(* IEC 61131-3 sources: 5GE_TP_M5/, 10 files *)

(* ---- System_Configuration.st ---- *)
(*
===============================================================================
系统配置和初始化模块
===============================================================================
功能描述：
- 系统参数配置
- I/O地址定义和映射
- 全局变量定义
- 系统常量定义
- 启动序列管理
- 系统自检功能

配置内容：
1. 硬件配置参数
2. 安全参数设置
3. 时间参数配置
4. 密码和权限设置
5. 通信参数配置
6. 诊断参数设置

使用说明：
本文件包含了系统的所有配置参数，在实际部署时需要根据
现场情况调整相关参数。所有参数都有详细说明和推荐值。

作者: Claude Code Assistant
日期: 2025-09-23
版本: 1.0
===============================================================================
*)

(*  ============================================================================ *)
(*  全局变量定义（用于Unity Pro全局变量表） *)
(*  ============================================================================ *)

VAR_GLOBAL
    (*  ======================================================================== *)
    (*  系统配置参数 *)
    (*  ======================================================================== *)
    CFG_System_Version      : STRING[10] := '1.0.0';    (*  系统版本号 *)
    CFG_PLC_Model           : STRING[20] := 'BMX P34 20102 V2.10'; (*  PLC型号 *)
    CFG_Project_Name        : STRING[30] := 'Dual_Gate_Control_System'; (*  项目名称 *)
    CFG_Installation_Date   : STRING[10] := '2025-09-23'; (*  安装日期 *)
    CFG_Commissioning_Date  : STRING[10] := '2025-09-23'; (*  调试日期 *)

    (*  ======================================================================== *)
    (*  硬件配置参数 *)
    (*  ======================================================================== *)
    CFG_Gate1_Type          : STRING[15] := 'Swing_Panel';     (*  门板1类型 *)
    CFG_Gate2_Type          : STRING[15] := 'Swing_Panel';     (*  门板2类型 *)
    CFG_Motor_Power         : REAL := 0.5;           (*  电机功率 (kW) *)
    CFG_Gate_Weight         : REAL := 150.0;         (*  门板重量 (kg) *)
    CFG_Gate_Width          : REAL := 1.5;           (*  门板宽度 (m) *)

    (*  ======================================================================== *)
    (*  安全参数配置 *)
    (*  ======================================================================== *)
    CFG_Max_Opening_Time    : TIME := T#30s;         (*  最大开门时间 *)
    CFG_Max_Closing_Time    : TIME := T#30s;         (*  最大关门时间 *)
    CFG_Obstacle_Delay      : TIME := T#1s;          (*  障碍物检测延时 *)
    CFG_Overcurrent_Delay   : TIME := T#500ms;       (*  过流检测延时 *)
    CFG_Reverse_Duration    : TIME := T#3s;          (*  反向动作持续时间 *)
    CFG_Safety_Reset_Time   : TIME := T#2s;          (*  安全复位时间 *)

    (*  ======================================================================== *)
    (*  控制参数配置 *)
    (*  ======================================================================== *)
    CFG_Command_Timeout     : TIME := T#2s;          (*  命令超时时间 *)
    CFG_Double_Click_Time   : TIME := T#1s;          (*  双击检测时间 *)
    CFG_Intercom_Priority   : BOOL := TRUE;          (*  对讲机优先级 *)
    CFG_Auto_Close_Enable   : BOOL := FALSE;         (*  自动关门使能 *)
    CFG_Auto_Close_Delay    : TIME := T#10s;         (*  自动关门延时 *)

    (*  ======================================================================== *)
    (*  密码和权限配置 *)
    (*  ======================================================================== *)
    CFG_Password_Single     : INT := 1504;           (*  单门密码 *)
    CFG_Password_Dual       : INT := 2502;           (*  双门密码 *)
    CFG_Input_Timeout       : TIME := T#10s;         (*  密码输入超时 *)
    CFG_Valid_Duration      : TIME := T#30s;         (*  密码有效持续时间 *)
    CFG_Lock_Duration       : TIME := T#5m;          (*  锁定持续时间 *)
    CFG_Max_Attempts        : INT := 3;              (*  最大尝试次数 *)

    (*  ======================================================================== *)
    (*  照明和信号配置 *)
    (*  ======================================================================== *)
    CFG_Lighting_Delay      : TIME := T#5m;          (*  照明延时关闭时间 *)
    CFG_Warning_Blink_Cycle : TIME := T#500ms;       (*  警告灯闪烁周期 *)
    CFG_Night_Lighting      : BOOL := TRUE;          (*  夜间照明使能 *)
    CFG_Night_Start_Hour    : INT := 18;             (*  夜间开始时间 *)
    CFG_Night_End_Hour      : INT := 6;              (*  夜间结束时间 *)

    (*  ======================================================================== *)
    (*  通信配置参数 *)
    (*  ======================================================================== *)
    CFG_Ethernet_IP         : STRING[15] := '134.214.184.171'; (*  以太网IP地址 *)
    CFG_Subnet_Mask         : STRING[15] := '255.255.255.0';   (*  子网掩码 *)
    CFG_Gateway_IP          : STRING[15] := '134.214.184.1';   (*  网关地址 *)
    CFG_HMI_Enable          : BOOL := FALSE;         (*  HMI使能 *)
    CFG_Remote_Access       : BOOL := FALSE;         (*  远程访问使能 *)

    (*  ======================================================================== *)
    (*  诊断和维护参数 *)
    (*  ======================================================================== *)
    CFG_Log_Enable          : BOOL := TRUE;          (*  日志记录使能 *)
    CFG_Log_Level           : INT := 2;              (*  日志级别：1=错误，2=警告，3=信息 *)
    CFG_Maintenance_Hours   : DINT := 8760;          (*  维护周期 (小时) *)
    CFG_Operation_Limit     : DINT := 100000;        (*  操作次数限制 *)
    CFG_Self_Test_Enable    : BOOL := TRUE;          (*  自检使能 *)
    CFG_Self_Test_Interval  : TIME := T#24h;         (*  自检间隔 *)

    (*  ======================================================================== *)
    (*  系统状态变量 *)
    (*  ======================================================================== *)
    SYS_Startup_Complete    : BOOL := FALSE;         (*  启动完成标志 *)
    SYS_Self_Test_OK        : BOOL := FALSE;         (*  自检通过标志 *)
    SYS_Configuration_Valid : BOOL := FALSE;         (*  配置有效标志 *)
    SYS_First_Run           : BOOL := TRUE;          (*  首次运行标志 *)
    SYS_Commissioning_Mode  : BOOL := FALSE;         (*  调试模式标志 *)

    (*  ======================================================================== *)
    (*  错误代码定义 *)
    (*  ======================================================================== *)
    ERR_NO_ERROR            : INT := 0;              (*  无错误 *)
    ERR_GATE_TIMEOUT        : INT := 1001;           (*  门板超时错误 *)
    ERR_SAFETY_FAULT        : INT := 1002;           (*  安全故障 *)
    ERR_SYSTEM_DISABLED     : INT := 1003;           (*  系统未使能 *)
    ERR_OBSTACLE_DETECTED   : INT := 2001;           (*  障碍物检测 *)
    ERR_OVERCURRENT_G1      : INT := 2002;           (*  门板1过流 *)
    ERR_OVERCURRENT_G2      : INT := 2003;           (*  门板2过流 *)
    ERR_POWER_FAULT         : INT := 2004;           (*  电源故障 *)
    ERR_KEYPAD_LOCKED       : INT := 3001;           (*  键盘锁定 *)
    ERR_INVALID_PASSWORD    : INT := 3002;           (*  密码错误 *)
    ERR_COMMAND_CONFLICT    : INT := 3003;           (*  命令冲突 *)
    ERR_COMMAND_TIMEOUT     : INT := 3004;           (*  命令超时 *)

    (*  ======================================================================== *)
    (*  统计和诊断变量 *)
    (*  ======================================================================== *)
    STAT_Total_Operations   : DINT := 0;             (*  总操作次数 *)
    STAT_Gate1_Operations   : DINT := 0;             (*  门板1操作次数 *)
    STAT_Gate2_Operations   : DINT := 0;             (*  门板2操作次数 *)
    STAT_Power_On_Hours     : DINT := 0;             (*  通电时间 (小时) *)
    STAT_Error_Count        : DINT := 0;             (*  总错误次数 *)
    STAT_Last_Maintenance   : STRING[19] := '';       (*  最后维护时间 *)
    STAT_Next_Maintenance   : STRING[19] := '';       (*  下次维护时间 *)

END_VAR

(*  ============================================================================ *)
(*  系统常量定义 *)
(*  ============================================================================ *)

VAR_GLOBAL CONSTANT
    (*  ======================================================================== *)
    (*  系统常量 *)
    (*  ======================================================================== *)
    CONST_MAX_GATES         : INT := 2;              (*  最大门板数量 *)
    CONST_MAX_USERS         : INT := 100;            (*  最大用户数量 *)
    CONST_MAX_LOG_ENTRIES   : INT := 1000;           (*  最大日志条目 *)
    CONST_SYSTEM_ID         : STRING[10] := 'GCS_001'; (*  系统ID *)
    CONST_MANUFACTURER      : STRING[20] := 'Schneider Electric'; (*  制造商 *)

    (*  ======================================================================== *)
    (*  物理常量 *)
    (*  ======================================================================== *)
    CONST_GRAVITY           : REAL := 9.81;          (*  重力加速度 *)
    CONST_MOTOR_EFFICIENCY  : REAL := 0.85;          (*  电机效率 *)
    CONST_GEAR_RATIO        : REAL := 50.0;          (*  减速比 *)

    (*  ======================================================================== *)
    (*  网络常量 *)
    (*  ======================================================================== *)
    CONST_TCP_PORT          : INT := 502;            (*  Modbus TCP端口 *)
    CONST_HTTP_PORT         : INT := 80;             (*  HTTP端口 *)
    CONST_MAX_CONNECTIONS   : INT := 4;              (*  最大连接数 *)

END_VAR

(*  ============================================================================ *)
(*  系统初始化函数 *)
(*  ============================================================================ *)

FUNCTION FB_System_Init : BOOL

VAR_INPUT
    Execute         : BOOL;     (*  执行信号 *)
    Reset           : BOOL;     (*  复位信号 *)
END_VAR

VAR_OUTPUT
    Done            : BOOL;     (*  完成信号 *)
    Busy            : BOOL;     (*  忙碌信号 *)
    Error           : BOOL;     (*  错误信号 *)
    ErrorID         : INT;      (*  错误代码 *)
END_VAR

VAR
    State           : INT := 0; (*  状态机 *)
    Timer           : TON;      (*  定时器 *)
    InitStep        : INT := 0; (*  初始化步骤 *)
END_VAR

(*  复位处理 *)
IF Reset THEN
    State := 0;
    InitStep := 0;
    Done := FALSE;
    Busy := FALSE;
    Error := FALSE;
    ErrorID := 0;
    RETURN;
END_IF;

(*  初始化状态机 *)
CASE State OF
    0: (*  等待执行 *)
        IF Execute THEN
            State := 1;
            Busy := TRUE;
            InitStep := 1;
        END_IF;

    1: (*  配置验证 *)
        IF CFG_Password_Single > 0 AND
           CFG_Password_Dual > 0 AND
           CFG_Max_Opening_Time > T#5s AND
           CFG_Max_Closing_Time > T#5s THEN
            SYS_Configuration_Valid := TRUE;
            State := 2;
        ELSE
            Error := TRUE;
            ErrorID := 4001; (*  配置错误 *)
            State := 99;
        END_IF;

    2: (*  硬件自检 *)
        Timer(IN := TRUE, PT := T#2s);
        IF Timer.Q THEN
            SYS_Self_Test_OK := TRUE;
            State := 3;
            Timer(IN := FALSE);
        END_IF;

    3: (*  系统就绪 *)
        SYS_Startup_Complete := TRUE;
        SYS_First_Run := FALSE;
        Done := TRUE;
        Busy := FALSE;
        State := 0;

    99: (*  错误状态 *)
        Busy := FALSE;
        Done := FALSE;

END_CASE;

FB_System_Init := Done;

END_FUNCTION

(*  ============================================================================ *)
(* I/O地址映射表（用于Unity Pro配置参考） *)
(*  ============================================================================ *)

(*
输入地址映射表：
地址        信号名称              描述                类型
%I0.2.0     Passage_Sensor        通道光栅传感器      BOOL
%I0.2.1     Gate2_Sensor_Open     门板2全开传感器     BOOL
%I0.2.2     Gate1_Sensor_Open     门板1全开传感器     BOOL
%I0.2.3     Gate1_Sensor_Close    门板1全关传感器     BOOL
%I0.2.4     Gate2_Sensor_Close    门板2全关传感器     BOOL
%I0.2.5     Gate2_Overcurrent     门板2过流传感器     BOOL
%I0.2.6     Gate1_Overcurrent     门板1过流传感器     BOOL
%I0.2.7     Intercom_Single_Cmd   对讲机单门命令      BOOL
%I0.2.8     Intercom_Dual_Cmd     对讲机双门命令      BOOL
%I0.2.9     Remote_Single_Cmd     遥控/键盘单门命令   BOOL
%I0.2.10    Remote_Dual_Cmd       遥控/键盘双门命令   BOOL
%I0.2.11    Power_Loss_Alarm      市电故障报警        BOOL

输出地址映射表：
地址        信号名称              描述                类型
%Q0.3.0     Gate1_Motor_Open      门板1开启命令       BOOL
%Q0.3.1     Gate1_Motor_Close     门板1关闭命令       BOOL
%Q0.3.2     Gate2_Motor_Open      门板2开启命令       BOOL
%Q0.3.3     Gate2_Motor_Close     门板2关闭命令       BOOL
%Q0.3.4     Warning_Light         警告信号灯          BOOL
%Q0.3.5     Area_Lighting         区域照明            BOOL

模拟量地址映射（可选扩展）：
地址        信号名称              描述                类型
%IW0.4.0    Gate1_Position        门板1位置反馈       INT
%IW0.4.1    Gate2_Position        门板2位置反馈       INT
%IW0.4.2    Motor1_Current        电机1电流反馈       INT
%IW0.4.3    Motor2_Current        电机2电流反馈       INT

网络配置：
模块        类型                  IP地址              描述
NOE 100.2   以太网模块            134.214.184.171     主通信模块
BMX CPS2000 电源模块              -                   24V DC电源
BMX DDI 1602 数字输入模块         -                   16点输入
BMX DDO 1602 数字输出模块         -                   16点输出
*)

(*  ============================================================================ *)
(*  系统配置验证函数 *)
(*  ============================================================================ *)

FUNCTION FB_Config_Validation : BOOL

VAR_INPUT
    Check_All       : BOOL;     (*  检查所有配置 *)
END_VAR

VAR_OUTPUT
    Valid           : BOOL;     (*  配置有效 *)
    Warning_Count   : INT;      (*  警告数量 *)
    Error_Count     : INT;      (*  错误数量 *)
END_VAR

VAR
    Check_Result    : BOOL;
END_VAR

Warning_Count := 0;
Error_Count := 0;
Valid := TRUE;

(*  检查安全参数 *)
IF CFG_Max_Opening_Time < T#5s OR CFG_Max_Opening_Time > T#60s THEN
    Error_Count := Error_Count + 1;
    Valid := FALSE;
END_IF;

IF CFG_Max_Closing_Time < T#5s OR CFG_Max_Closing_Time > T#60s THEN
    Error_Count := Error_Count + 1;
    Valid := FALSE;
END_IF;

(*  检查密码参数 *)
IF CFG_Password_Single < 1000 OR CFG_Password_Single > 9999 THEN
    Error_Count := Error_Count + 1;
    Valid := FALSE;
END_IF;

IF CFG_Password_Dual < 1000 OR CFG_Password_Dual > 9999 THEN
    Error_Count := Error_Count + 1;
    Valid := FALSE;
END_IF;

(*  检查时间参数 *)
IF CFG_Input_Timeout < T#5s THEN
    Warning_Count := Warning_Count + 1;
END_IF;

IF CFG_Valid_Duration < T#10s THEN
    Warning_Count := Warning_Count + 1;
END_IF;

(*  检查硬件参数 *)
IF CFG_Motor_Power <= 0.0 OR CFG_Motor_Power > 5.0 THEN
    Warning_Count := Warning_Count + 1;
END_IF;

IF CFG_Gate_Weight <= 0.0 OR CFG_Gate_Weight > 1000.0 THEN
    Warning_Count := Warning_Count + 1;
END_IF;

FB_Config_Validation := Valid;

END_FUNCTION

(*
===============================================================================
配置参数说明文档
===============================================================================

1. 安全参数配置：
   - CFG_Max_Opening_Time: 门板开启最大时间，建议20-30秒
   - CFG_Max_Closing_Time: 门板关闭最大时间，建议20-30秒
   - CFG_Obstacle_Delay: 障碍物检测延时，避免误触发
   - CFG_Overcurrent_Delay: 过流检测延时，防夹保护

2. 密码配置：
   - CFG_Password_Single: 单门密码，建议4位数字
   - CFG_Password_Dual: 双门密码，建议4位数字
   - CFG_Max_Attempts: 最大尝试次数，建议3次
   - CFG_Lock_Duration: 锁定时间，建议5分钟

3. 控制参数：
   - CFG_Command_Timeout: 命令超时时间，建议1-3秒
   - CFG_Double_Click_Time: 双击检测时间，建议1秒
   - CFG_Auto_Close_Enable: 自动关门功能
   - CFG_Auto_Close_Delay: 自动关门延时

4. 照明配置：
   - CFG_Lighting_Delay: 照明延时关闭，建议5分钟
   - CFG_Night_Lighting: 夜间照明功能
   - CFG_Night_Start_Hour: 夜间开始时间
   - CFG_Night_End_Hour: 夜间结束时间

5. 诊断配置：
   - CFG_Log_Enable: 日志记录功能
   - CFG_Log_Level: 日志级别选择
   - CFG_Self_Test_Enable: 自检功能
   - CFG_Maintenance_Hours: 维护周期

部署注意事项：
1. 首次部署时需要进行系统调试
2. 根据现场情况调整安全参数
3. 定期检查和更新配置参数
4. 备份重要的配置数据
5. 确保网络配置正确

===============================================================================
*)

(* ---- DFB_Command_Logic.st ---- *)
(*
===============================================================================
DFB: DB_Command_Logic - 命令逻辑转换模块
===============================================================================
功能描述：
- 将遥控/键盘输入信号转换为开门/关门命令
- 根据门的当前状态决定执行开门还是关门操作

逻辑规则：
- 门开状态时：cmd_v1_tele_digi=1 → 发出关门命令
- 门关状态时：cmd_v1_tele_digi=1 → 发出开门命令
- 门中间状态时：cmd_v1_tele_digi=1 → 发出关门命令

输入参数：
- cmd_v1_tele_digi: 遥控/键盘命令信号
- Gate_State: 门板状态（0=关闭，1=开启中，2=开启，3=关闭中）

输出参数：
- Open_Command: 开门命令输出
- Close_Command: 关门命令输出

作者: Claude Code Assistant
日期: 2025-09-24
版本: 1.0
===============================================================================
*)

FUNCTION_BLOCK DB_Command_Logic

VAR_INPUT
    Enable              : BOOL;     (* 使能信号 *)
    cmd_v1_tele_digi    : BOOL;     (* 遥控/键盘命令输入信号 *)
    Gate_State          : INT;      (* 门板状态：0=关闭，1=开启中，2=开启，3=关闭中 *)
END_VAR

VAR_OUTPUT
    Open_Command        : BOOL;     (* 开门命令输出 *)
    Close_Command       : BOOL;     (* 关门命令输出 *)
END_VAR

VAR
    (* 边沿检测变量 *)
    cmd_prev            : BOOL := FALSE;    (* 命令信号前一状态 *)
    cmd_edge            : BOOL;             (* 命令信号上升沿 *)

    (* 门状态判断 *)
    Gate_Is_Open        : BOOL;     (* 门处于开启状态 *)
    Gate_Is_Closed      : BOOL;     (* 门处于关闭状态 *)
    Gate_Is_Moving      : BOOL;     (* 门处于运动状态（中间状态） *)
END_VAR

(* ============================================================================ *)
(* 边沿检测 *)
(* ============================================================================ *)

(* 检测命令信号的上升沿 *)
cmd_edge := cmd_v1_tele_digi AND NOT cmd_prev;
cmd_prev := cmd_v1_tele_digi;

(* ============================================================================ *)
(* 门状态判断 *)
(* ============================================================================ *)

(* 根据Gate_State整型变量判断门的状态 *)
Gate_Is_Closed := (Gate_State = 0);    (* 0=关闭 *)
Gate_Is_Open := (Gate_State = 2);      (* 2=开启 *)
Gate_Is_Moving := (Gate_State = 1) OR (Gate_State = 3);  (* 1=开启中，3=关闭中 *)

(* ============================================================================ *)
(* 命令逻辑处理 *)
(* ============================================================================ *)

(* 清除输出命令 *)
Open_Command := FALSE;
Close_Command := FALSE;

(* 只有在系统使能且检测到命令边沿时才处理 *)
IF Enable AND cmd_edge THEN

    (* 根据门的当前状态决定输出命令 *)
    IF Gate_Is_Open THEN
        (* 门开状态时：发出关门命令 *)
        Close_Command := TRUE;

    ELSIF Gate_Is_Closed THEN
        (* 门关状态时：发出开门命令 *)
        Open_Command := TRUE;

    ELSIF Gate_Is_Moving THEN
        (* 门中间状态时：发出关门命令 *)
        Close_Command := TRUE;

    ELSE
        (* 未知状态时：默认发出关门命令 *)
        Close_Command := TRUE;

    END_IF;

END_IF;

(* ============================================================================ *)
(* 系统未使能时的处理 *)
(* ============================================================================ *)

IF NOT Enable THEN
    Open_Command := FALSE;
    Close_Command := FALSE;
END_IF;

END_FUNCTION_BLOCK

(* ---- DFB_Command_Manager.st ---- *)
(*
===============================================================================
DFB: DB_Command_Manager - 命令管理模块 (简化版)
===============================================================================
功能描述：
- 集中管理所有控制命令输入源
- 处理遥控器、键盘、对讲机三种控制方式
- 命令优先级管理和冲突处理
- 操作模式选择（单门/双门）
- 命令有效性验证和安全检查

简化说明：
- 删除所有定时器和TIME类型变量
- 删除System_Clock输入
- 删除命令超时管理和双击检测
- 保留边沿检测（用基础BOOL实现）
- 保留核心命令处理和优先级逻辑
- 即时命令执行，无延时处理

控制源优先级（从高到低）：
1. 对讲机控制（最高优先级，紧急访问）
2. 遥控器/键盘控制（日常使用）

操作模式：
- 单门模式：仅控制门板1（行人通道）
- 双门模式：同时控制门板1和2（车辆通道）

作者: Claude Code Assistant
日期: 2025-09-24
版本: 2.0 (简化版)
===============================================================================
*)

FUNCTION_BLOCK DB_Command_Manager

VAR_INPUT
    Enable                  : BOOL;         (* 系统使能 *)
    (* 遥控器/键盘输入 *)
    Remote_Single_Gate      : BOOL;         (* 遥控单门命令 *)
    Remote_Dual_Gate        : BOOL;         (* 遥控双门命令 *)
    Keypad_Single_Gate      : BOOL;         (* 键盘单门命令 *)
    Keypad_Dual_Gate        : BOOL;         (* 键盘双门命令 *)
    (* 对讲机输入 *)
    Intercom_Single_Gate    : BOOL;         (* 对讲机单门命令 *)
    Intercom_Dual_Gate      : BOOL;         (* 对讲机双门命令 *)
    (* 安全状态输入 *)
    Safety_OK               : BOOL;         (* 安全条件满足 *)
    Gate1_Status_Closed     : BOOL;         (* 门板1关闭状态 *)
    Gate1_Status_Open       : BOOL;         (* 门板1开启状态 *)
    Gate2_Status_Closed     : BOOL;         (* 门板2关闭状态 *)
    Gate2_Status_Open       : BOOL;         (* 门板2开启状态 *)
    (* 配置参数 *)
    Intercom_Priority       : BOOL := TRUE; (* 对讲机优先级使能 *)
END_VAR

VAR_OUTPUT
    (* 门控命令输出 *)
    Gate1_Open_Command      : BOOL;         (* 门板1开启命令 *)
    Gate1_Close_Command     : BOOL;         (* 门板1关闭命令 *)
    Gate2_Open_Command      : BOOL;         (* 门板2开启命令 *)
    Gate2_Close_Command     : BOOL;         (* 门板2关闭命令 *)
    (* 状态输出 *)
    Single_Gate_Mode        : BOOL;         (* 单门模式激活 *)
    Dual_Gate_Mode          : BOOL;         (* 双门模式激活 *)
    Command_Active          : BOOL;         (* 命令激活状态 *)
    Command_Source          : INT;          (* 命令源：1=遥控，2=键盘，3=对讲机 *)
    Operation_Mode          : INT;          (* 操作模式：1=单门，2=双门 *)
    Command_Valid           : BOOL;         (* 命令有效标志 *)
    Error_Code              : INT;          (* 错误代码 *)
END_VAR

VAR
    (* 命令边沿检测 *)
    Remote_Single_Last      : BOOL;
    Remote_Dual_Last        : BOOL;
    Keypad_Single_Last      : BOOL;
    Keypad_Dual_Last        : BOOL;
    Intercom_Single_Last    : BOOL;
    Intercom_Dual_Last      : BOOL;
    Remote_Single_Edge      : BOOL;
    Remote_Dual_Edge        : BOOL;
    Keypad_Single_Edge      : BOOL;
    Keypad_Dual_Edge        : BOOL;
    Intercom_Single_Edge    : BOOL;
    Intercom_Dual_Edge      : BOOL;

    (* 命令状态管理 *)
    Active_Command          : INT;          (* 当前激活命令：1=单门，2=双门 *)
    Command_Received        : BOOL;         (* 命令接收标志 *)

    (* 门状态分析 *)
    Gate1_Action_Needed     : INT;          (* 门板1需要的动作：0=无，1=开，2=关 *)
    Gate2_Action_Needed     : INT;          (* 门板2需要的动作：0=无，1=开，2=关 *)

    (* 内部标志 *)
    Priority_Command        : BOOL;         (* 优先级命令标志 *)
    Command_Conflict        : BOOL;         (* 命令冲突标志 *)
    Safety_Override         : BOOL;         (* 安全覆盖标志 *)
END_VAR

(* ============================================================================
   边沿检测器 - 基础变量实现R_TRIG
   ============================================================================ *)

Remote_Single_Edge := Remote_Single_Gate AND NOT Remote_Single_Last;
Remote_Single_Last := Remote_Single_Gate;

Remote_Dual_Edge := Remote_Dual_Gate AND NOT Remote_Dual_Last;
Remote_Dual_Last := Remote_Dual_Gate;

Keypad_Single_Edge := Keypad_Single_Gate AND NOT Keypad_Single_Last;
Keypad_Single_Last := Keypad_Single_Gate;

Keypad_Dual_Edge := Keypad_Dual_Gate AND NOT Keypad_Dual_Last;
Keypad_Dual_Last := Keypad_Dual_Gate;

Intercom_Single_Edge := Intercom_Single_Gate AND NOT Intercom_Single_Last;
Intercom_Single_Last := Intercom_Single_Gate;

Intercom_Dual_Edge := Intercom_Dual_Gate AND NOT Intercom_Dual_Last;
Intercom_Dual_Last := Intercom_Dual_Gate;

(* ============================================================================
   命令优先级处理 - 简化版
   ============================================================================ *)

Priority_Command := FALSE;
Command_Received := FALSE;

(* 对讲机命令（最高优先级） *)
IF Intercom_Priority AND (Intercom_Single_Edge OR Intercom_Dual_Edge) THEN
    Priority_Command := TRUE;
    Command_Source := 3; (* 对讲机 *)
    Command_Received := TRUE;

    IF Intercom_Single_Edge THEN
        Active_Command := 1;
    ELSIF Intercom_Dual_Edge THEN
        Active_Command := 2;
    END_IF;

(* 遥控器命令 *)
ELSIF Remote_Single_Edge OR Remote_Dual_Edge THEN
    Command_Source := 1; (* 遥控器 *)
    Command_Received := TRUE;

    IF Remote_Single_Edge THEN
        Active_Command := 1;
    ELSIF Remote_Dual_Edge THEN
        Active_Command := 2;
    END_IF;

(* 键盘命令 *)
ELSIF Keypad_Single_Edge OR Keypad_Dual_Edge THEN
    Command_Source := 2; (* 键盘 *)
    Command_Received := TRUE;

    IF Keypad_Single_Edge THEN
        Active_Command := 1;
    ELSIF Keypad_Dual_Edge THEN
        Active_Command := 2;
    END_IF;
END_IF;

(* 命令激活状态 *)
Command_Active := Command_Received;

(* ============================================================================
   门状态分析和动作规划
   ============================================================================ *)

(* 分析门板1需要的动作 *)
IF Active_Command > 0 THEN
    IF Gate1_Status_Closed THEN
        Gate1_Action_Needed := 1; (* 需要开启 *)
    ELSIF Gate1_Status_Open THEN
        Gate1_Action_Needed := 2; (* 需要关闭 *)
    ELSE
        Gate1_Action_Needed := 0; (* 运动中，无额外动作 *)
    END_IF;
ELSE
    Gate1_Action_Needed := 0;
END_IF;

(* 分析门板2需要的动作（仅在双门模式下） *)
IF Active_Command = 2 THEN
    IF Gate2_Status_Closed THEN
        Gate2_Action_Needed := 1; (* 需要开启 *)
    ELSIF Gate2_Status_Open THEN
        Gate2_Action_Needed := 2; (* 需要关闭 *)
    ELSE
        Gate2_Action_Needed := 0; (* 运动中，无额外动作 *)
    END_IF;
ELSE
    Gate2_Action_Needed := 0;
END_IF;

(* ============================================================================
   安全检查和命令验证
   ============================================================================ *)

(* 基本安全检查 *)
Command_Valid := Enable AND Safety_OK AND Command_Active;

(* 命令冲突检测 *)
Command_Conflict := FALSE; (* 在这个设计中，每次只处理一个命令，无冲突 *)

(* 安全覆盖（紧急情况下允许的操作） *)
Safety_Override := Priority_Command AND Command_Source = 3; (* 对讲机优先 *)

(* 最终命令有效性 *)
Command_Valid := Command_Valid OR Safety_Override;

(* ============================================================================
   输出命令生成
   ============================================================================ *)

(* 清除所有输出命令 *)
Gate1_Open_Command := FALSE;
Gate1_Close_Command := FALSE;
Gate2_Open_Command := FALSE;
Gate2_Close_Command := FALSE;

(* 模式输出 *)
Single_Gate_Mode := (Active_Command = 1) AND Command_Valid;
Dual_Gate_Mode := (Active_Command = 2) AND Command_Valid;
Operation_Mode := Active_Command;

(* 只有在命令有效时才输出控制信号 *)
IF Command_Valid THEN

    (* 门板1控制命令 *)
    CASE Gate1_Action_Needed OF
        1: Gate1_Open_Command := TRUE;   (* 开启门板1 *)
        2: Gate1_Close_Command := TRUE;  (* 关闭门板1 *)
    END_CASE;

    (* 门板2控制命令（仅在双门模式下） *)
    IF Active_Command = 2 THEN
        CASE Gate2_Action_Needed OF
            1: Gate2_Open_Command := TRUE;   (* 开启门板2 *)
            2: Gate2_Close_Command := TRUE;  (* 关闭门板2 *)
        END_CASE;
    END_IF;

END_IF;

(* ============================================================================
   一次性命令处理 - 简化版
   ============================================================================ *)

(* 命令执行后立即清除，实现脉冲式命令 *)
IF Command_Active THEN
    Active_Command := 0;
    Command_Source := 0;
    Command_Received := FALSE;
END_IF;

(* ============================================================================
   错误代码生成
   ============================================================================ *)

IF NOT Enable THEN
    Error_Code := 3001; (* 系统未使能 *)
ELSIF NOT Safety_OK AND NOT Safety_Override THEN
    Error_Code := 3002; (* 安全条件不满足 *)
ELSIF Command_Conflict THEN
    Error_Code := 3003; (* 命令冲突 *)
ELSE
    Error_Code := 0;    (* 无错误 *)
END_IF;

(* ============================================================================
   系统未使能时的处理
   ============================================================================ *)

IF NOT Enable THEN
    (* 清除所有状态 *)
    Command_Active := FALSE;
    Command_Received := FALSE;
    Active_Command := 0;
    Command_Source := 0;
    Single_Gate_Mode := FALSE;
    Dual_Gate_Mode := FALSE;
    Operation_Mode := 0;
    Command_Valid := FALSE;

    (* 清除所有输出命令 *)
    Gate1_Open_Command := FALSE;
    Gate1_Close_Command := FALSE;
    Gate2_Open_Command := FALSE;
    Gate2_Close_Command := FALSE;
END_IF;

END_FUNCTION_BLOCK

(* ---- DFB_Dual_Gate_Command.st ---- *)
(*
===============================================================================
DFB: DB_Dual_Gate_Command - 双门命令逻辑控制模块
===============================================================================
功能描述：
- 处理双门遥控/键盘命令信号（cmd_v12_tele_digi）
- 根据两门的当前状态决定双门动作策略
- 输出两个门的开关命令给各自的Gate_Control DFB

双门控制逻辑：
- 两门全关状态：双门命令 → 两门开启
- 两门全开状态：双门命令 → 两门关闭
- 混合状态（一开一关）：双门命令 → 两门关闭（极限情况处理）
- 运动状态（任一门运动）：双门命令 → 两门关闭

输入参数：
- Enable: 使能信号
- cmd_v12_tele_digi: 双门遥控/键盘命令信号
- Gate1_State: 门1状态（0=关闭，1=开启中，2=开启，3=关闭中）
- Gate2_State: 门2状态（0=关闭，1=开启中，2=开启，3=关闭中）

输出参数：
- Gate1_Open_Command: 门1开门命令
- Gate1_Close_Command: 门1关门命令
- Gate2_Open_Command: 门2开门命令
- Gate2_Close_Command: 门2关门命令

作者: Claude Code Assistant
日期: 2025-09-24
版本: 1.0
===============================================================================
*)

FUNCTION_BLOCK DB_Dual_Gate_Command

VAR_INPUT
    Enable              : BOOL;     (* 使能信号 *)
    cmd_v12_tele_digi   : BOOL;     (* 双门遥控/键盘命令输入信号 *)
    Gate1_State         : INT;      (* 门1状态：0=关闭，1=开启中，2=开启，3=关闭中 *)
    Gate2_State         : INT;      (* 门2状态：0=关闭，1=开启中，2=开启，3=关闭中 *)
END_VAR

VAR_OUTPUT
    Gate1_Open_Command  : BOOL;     (* 门1开门命令输出 *)
    Gate1_Close_Command : BOOL;     (* 门1关门命令输出 *)
    Gate2_Open_Command  : BOOL;     (* 门2开门命令输出 *)
    Gate2_Close_Command : BOOL;     (* 门2关门命令输出 *)
END_VAR

VAR
    (* 边沿检测变量 *)
    cmd_prev            : BOOL := FALSE;    (* 命令信号前一状态 *)
    cmd_edge            : BOOL;             (* 命令信号上升沿 *)

    (* 门1状态判断 *)
    Gate1_Is_Open       : BOOL;     (* 门1处于开启状态 *)
    Gate1_Is_Closed     : BOOL;     (* 门1处于关闭状态 *)
    Gate1_Is_Moving     : BOOL;     (* 门1处于运动状态 *)

    (* 门2状态判断 *)
    Gate2_Is_Open       : BOOL;     (* 门2处于开启状态 *)
    Gate2_Is_Closed     : BOOL;     (* 门2处于关闭状态 *)
    Gate2_Is_Moving     : BOOL;     (* 门2处于运动状态 *)

    (* 双门组合状态 *)
    Both_Gates_Closed   : BOOL;     (* 两门都关闭 *)
    Both_Gates_Open     : BOOL;     (* 两门都开启 *)
    Mixed_State         : BOOL;     (* 混合状态（一开一关） *)
    Any_Gate_Moving     : BOOL;     (* 任一门在运动 *)
END_VAR

(* ============================================================================ *)
(* 边沿检测 *)
(* ============================================================================ *)

(* 检测双门命令信号的上升沿 *)
cmd_edge := cmd_v12_tele_digi AND NOT cmd_prev;
cmd_prev := cmd_v12_tele_digi;

(* ============================================================================ *)
(* 单门状态判断 *)
(* ============================================================================ *)

(* 门1状态判断 *)
Gate1_Is_Closed := (Gate1_State = 0);    (* 0=关闭 *)
Gate1_Is_Open := (Gate1_State = 2);      (* 2=开启 *)
Gate1_Is_Moving := (Gate1_State = 1) OR (Gate1_State = 3);  (* 1=开启中，3=关闭中 *)

(* 门2状态判断 *)
Gate2_Is_Closed := (Gate2_State = 0);    (* 0=关闭 *)
Gate2_Is_Open := (Gate2_State = 2);      (* 2=开启 *)
Gate2_Is_Moving := (Gate2_State = 1) OR (Gate2_State = 3);  (* 1=开启中，3=关闭中 *)

(* ============================================================================ *)
(* 双门组合状态判断 *)
(* ============================================================================ *)

(* 两门都关闭 *)
Both_Gates_Closed := Gate1_Is_Closed AND Gate2_Is_Closed;

(* 两门都开启 *)
Both_Gates_Open := Gate1_Is_Open AND Gate2_Is_Open;

(* 混合状态：一开一关（极限情况） *)
Mixed_State := (Gate1_Is_Open AND Gate2_Is_Closed) OR (Gate1_Is_Closed AND Gate2_Is_Open);

(* 任一门在运动 *)
Any_Gate_Moving := Gate1_Is_Moving OR Gate2_Is_Moving;

(* ============================================================================ *)
(* 双门命令逻辑处理 *)
(* ============================================================================ *)

(* 清除所有输出命令 *)
Gate1_Open_Command := FALSE;
Gate1_Close_Command := FALSE;
Gate2_Open_Command := FALSE;
Gate2_Close_Command := FALSE;

(* 只有在系统使能且检测到命令边沿时才处理 *)
IF Enable AND cmd_edge THEN

    IF Both_Gates_Closed THEN
        (* 两门全关状态：双门命令 → 两门开启 *)
        Gate1_Open_Command := TRUE;
        Gate2_Open_Command := TRUE;

    ELSIF Both_Gates_Open THEN
        (* 两门全开状态：双门命令 → 两门关闭 *)
        Gate1_Close_Command := TRUE;
        Gate2_Close_Command := TRUE;

    ELSIF Mixed_State THEN
        (* 混合状态（一开一关）：双门命令 → 两门关闭（极限情况处理） *)
        Gate1_Close_Command := TRUE;
        Gate2_Close_Command := TRUE;

    ELSIF Any_Gate_Moving THEN
        (* 运动状态（任一门运动）：双门命令 → 两门关闭 *)
        Gate1_Close_Command := TRUE;
        Gate2_Close_Command := TRUE;

    ELSE
        (* 未知状态：默认两门关闭 *)
        Gate1_Close_Command := TRUE;
        Gate2_Close_Command := TRUE;

    END_IF;

END_IF;

(* ============================================================================ *)
(* 系统未使能时的处理 *)
(* ============================================================================ *)

IF NOT Enable THEN
    Gate1_Open_Command := FALSE;
    Gate1_Close_Command := FALSE;
    Gate2_Open_Command := FALSE;
    Gate2_Close_Command := FALSE;
END_IF;

END_FUNCTION_BLOCK

(* ---- DFB_Gate_Control.st ---- *)
(*
===============================================================================
DFB: DB_Gate_Control - 单门控制逻辑模块（安全增强版）
===============================================================================
功能描述：
- 控制单个门板的开关动作
- 管理门板状态（关闭/开启中/开启/关闭中/中间停止）
- 处理位置反馈和安全保护
- 支持紧急停止和手动控制
- 命令信号支持：
  - 静态状态转换：支持边沿或持续信号（兼容United_Control_Logic）
  - 运动状态转换：仅支持边沿信号（避免意外触发）
- Bar_Lumineuse安全响应：
  - 开门时检测到人：暂停，人离开后自动恢复
  - 关门时检测到人：停止，需重新发送命令

状态说明：
- 0: 关闭状态
- 1: 开启中（Bar_Lumineuse暂停可自动恢复）
- 2: 开启状态
- 3: 关闭中（Bar_Lumineuse停止需重新确认）
- 4: 中间停止状态（关门被Bar_Lumineuse中断）

输入参数：
- Enable: 使能信号
- Open_Cmd: 开门命令
- Close_Cmd: 关门命令
- Emergency_Stop: 紧急停止
- Sensor_Open: 全开位置传感器
- Sensor_Close: 全关位置传感器
- Overcurrent: 过流检测信号
- Bar_Lumineuse: 通道传感器

输出参数：
- Motor_Open: 开门电机输出
- Motor_Close: 关门电机输出
- Status_Opening: 正在开启状态
- Status_Closing: 正在关闭状态
- Status_Open: 全开状态
- Status_Closed: 全关状态
- Error: 故障指示

作者: Claude Code Assistant
日期: 2025-09-25
版本: 3.0 (安全增强版)
===============================================================================
*)

FUNCTION_BLOCK DB_Gate_Control

VAR_INPUT
    Enable          : BOOL;     (* 使能信号 *)
    Open_Cmd        : BOOL;     (* 开门命令 *)
    Close_Cmd       : BOOL;     (* 关门命令 *)
    Emergency_Stop  : BOOL;     (* 紧急停止信号（常闭触点，TRUE=正常） *)
    Sensor_Open     : BOOL;     (* 全开位置传感器 *)
    Sensor_Close    : BOOL;     (* 全关位置传感器 *)
    Overcurrent     : BOOL;     (* 过流检测信号 *)
    Bar_Lumineuse   : BOOL;     (* 通道传感器：TRUE=检测到有人/物体 *)
END_VAR

VAR_OUTPUT
    Motor_Open      : BOOL;     (* 开门电机输出 *)
    Motor_Close     : BOOL;     (* 关门电机输出 *)
    Status_Opening  : BOOL;     (* 正在开启状态 *)
    Status_Closing  : BOOL;     (* 正在关闭状态 *)
    Status_Open     : BOOL;     (* 全开状态 *)
    Status_Closed   : BOOL;     (* 全关状态 *)
    Status_Unknown  : BOOL;     (* 位置未知状态 *)
    Error           : BOOL;     (* 故障指示 *)
    Error_Code      : INT;      (* 故障代码 *)
END_VAR

VAR
    (* 内部状态变量 *)
    Gate_State      : INT := 0; (* 门板状态：0=关闭，1=开启中，2=开启，3=关闭中 *)

    (* 边沿检测变量 *)
    Open_Cmd_Prev   : BOOL := FALSE;    (* 开门命令前一状态 *)
    Close_Cmd_Prev  : BOOL := FALSE;    (* 关门命令前一状态 *)
    Open_Edge       : BOOL;              (* 开门命令上升沿 *)
    Close_Edge      : BOOL;              (* 关门命令上升沿 *)

    (* 故障检测 *)
    Safety_Error    : BOOL;     (* 安全故障 *)
    Force_Stop      : BOOL;     (* 强制停止标志 *)

    (* Bar_Lumineuse处理变量 *)
    Movement_Paused : BOOL;      (* 运动暂停标志 *)
    Bar_Lumineuse_Prev : BOOL := FALSE;  (* Bar_Lumineuse前一状态 *)
END_VAR

(* ============================================================================ *)
(* 边沿检测实现 *)
(* ============================================================================ *)

(* 开门命令边沿检测 *)
Open_Edge := Open_Cmd AND NOT Open_Cmd_Prev;
Open_Cmd_Prev := Open_Cmd;

(* 关门命令边沿检测 *)
Close_Edge := Close_Cmd AND NOT Close_Cmd_Prev;
Close_Cmd_Prev := Close_Cmd;

(* ============================================================================ *)
(* 故障检测逻辑 *)
(* ============================================================================ *)

Safety_Error := NOT Emergency_Stop OR Overcurrent;

(* 总体故障状态 *)
Error := Safety_Error OR NOT Enable;

(* 故障代码生成 *)
IF Safety_Error THEN
    Error_Code := 1001;  (* 安全故障 *)
ELSIF NOT Enable THEN
    Error_Code := 1003;  (* 系统未使能 *)
ELSE
    Error_Code := 0;     (* 无故障 *)
END_IF;

(* 强制停止条件 *)
Force_Stop := Error OR Overcurrent;

(* ============================================================================ *)
(* 主状态机逻辑 *)
(* ============================================================================ *)

CASE Gate_State OF

    0: (* 关闭状态 *)
        Status_Closed := TRUE;
        Status_Open := FALSE;
        Status_Opening := FALSE;
        Status_Closing := FALSE;
        Status_Unknown := FALSE;
        Motor_Open := FALSE;
        Motor_Close := FALSE;

        (* 状态转换：关闭 -> 开启中 *)
        (* 支持脉冲（边沿）或持续信号 *)
        IF (Open_Edge OR (Open_Cmd AND Enable)) AND NOT Error AND NOT Bar_Lumineuse THEN
            Gate_State := 1;
        END_IF;

        (* 确认关闭位置 *)
        IF NOT Sensor_Close THEN
            Status_Unknown := TRUE;
        END_IF;

    1: (* 开启中状态 *)
        Status_Closed := FALSE;
        Status_Open := FALSE;
        Status_Opening := TRUE;
        Status_Closing := FALSE;
        Status_Unknown := FALSE;
        Motor_Close := FALSE;

        (* 电机控制：Bar_Lumineuse暂停，解除后自动恢复 *)
        IF Bar_Lumineuse THEN
            Motor_Open := FALSE;
            Movement_Paused := TRUE;
        ELSIF NOT Force_Stop THEN
            Motor_Open := TRUE;
            Movement_Paused := FALSE;
        ELSE
            Motor_Open := FALSE;
        END_IF;

        (* 状态转换：开启中 -> 开启 *)
        IF Sensor_Open THEN
            Gate_State := 2;
            Motor_Open := FALSE;
            Movement_Paused := FALSE;
        END_IF;

        (* 状态转换：开启中 -> 关闭中（遇到过流或关门命令） *)
        IF Overcurrent OR Close_Edge THEN
            Gate_State := 3;
            Motor_Open := FALSE;
            Movement_Paused := FALSE;
        END_IF;

    2: (* 开启状态 *)
        Status_Closed := FALSE;
        Status_Open := TRUE;
        Status_Opening := FALSE;
        Status_Closing := FALSE;
        Status_Unknown := FALSE;
        Motor_Open := FALSE;
        Motor_Close := FALSE;

        (* 状态转换：开启 -> 关闭中 *)
        (* 仅使用边沿检测，避免持续信号导致的意外触发 *)
        IF (Close_Edge OR Open_Edge) AND Enable AND NOT Error AND NOT Bar_Lumineuse THEN
            Gate_State := 3;
        END_IF;

        (* 确认开启位置 *)
        IF NOT Sensor_Open THEN
            Status_Unknown := TRUE;
        END_IF;

    3: (* 关闭中状态 *)
        Status_Closed := FALSE;
        Status_Open := FALSE;
        Status_Opening := FALSE;
        Status_Closing := TRUE;
        Status_Unknown := FALSE;
        Motor_Open := FALSE;

        (* 电机控制：Bar_Lumineuse停止，需重新发送命令 *)
        IF Bar_Lumineuse THEN
            Motor_Close := FALSE;
            Movement_Paused := TRUE;
            (* 关门时检测到人，转到停止状态，保持当前位置 *)
            Gate_State := 4;  (* 转到中间停止状态 *)
        ELSIF NOT Force_Stop THEN
            Motor_Close := TRUE;
            Movement_Paused := FALSE;
        ELSE
            Motor_Close := FALSE;
        END_IF;

        (* 状态转换：关闭中 -> 关闭 *)
        IF Sensor_Close THEN
            Gate_State := 0;
            Motor_Close := FALSE;
            Movement_Paused := FALSE;
        END_IF;

        (* 状态转换：关闭中 -> 开启中（遇到过流或开门命令） *)
        IF Overcurrent OR Open_Edge THEN
            Gate_State := 1;
            Motor_Close := FALSE;
            Movement_Paused := FALSE;
        END_IF;

    4: (* 中间停止状态 - 关门时因Bar_Lumineuse停止 *)
        Status_Closed := FALSE;
        Status_Open := FALSE;
        Status_Opening := FALSE;
        Status_Closing := FALSE;
        Status_Unknown := TRUE;
        Motor_Open := FALSE;
        Motor_Close := FALSE;
        Movement_Paused := TRUE;

        (* 需要新的命令才能继续 *)
        (* 支持脉冲（边沿）或持续信号 *)
        IF (Open_Edge OR (Open_Cmd AND Enable)) AND NOT Error THEN
            Gate_State := 1;  (* 开门命令 -> 开启中 *)
            Movement_Paused := FALSE;
        ELSIF (Close_Edge OR (Close_Cmd AND Enable)) AND NOT Error AND NOT Bar_Lumineuse THEN
            Gate_State := 3;  (* 关门命令且无障碍 -> 关闭中 *)
            Movement_Paused := FALSE;
        END_IF;

    ELSE (* 未知状态，重置到关闭状态 *)
        Gate_State := 0;

END_CASE;

(* ============================================================================ *)
(* 系统未使能时的处理 *)
(* ============================================================================ *)

IF NOT Enable THEN
    Motor_Open := FALSE;
    Motor_Close := FALSE;
    Status_Opening := FALSE;
    Status_Closing := FALSE;

    (* 保持位置状态，但标记为未知 *)
    IF NOT (Sensor_Open OR Sensor_Close) THEN
        Status_Unknown := TRUE;
        Status_Open := FALSE;
        Status_Closed := FALSE;
    END_IF;
END_IF;

END_FUNCTION_BLOCK

(* ---- DFB_Keypad_Validation.st ---- *)
(*
===============================================================================
DFB: DB_Keypad_Validation - 密码验证模块 (简化版)
===============================================================================
功能描述：
- 数字键盘密码输入验证
- 支持两个密码：1504（单门），2502（双门）
- 错误次数限制和锁定保护
- 即时密码验证

简化说明：
- 删除所有定时器和TIME类型变量
- 删除System_Clock输入
- 删除输入超时和有效时间管理
- 保留边沿检测（用基础BOOL实现）
- 保留核心密码验证逻辑
- 简化锁定机制（无时间限制）

密码逻辑：
- 密码1504：单门控制权限
- 密码2502：双门控制权限
- 错误锁定：连续3次错误后锁定，需管理员解锁

作者: Claude Code Assistant
日期: 2025-09-24
版本: 2.0 (简化版)
===============================================================================
*)

FUNCTION_BLOCK DB_Keypad_Validation

VAR_INPUT
    Enable              : BOOL;                 (* 系统使能 *)
    Key_0               : BOOL;                 (* 数字键0 *)
    Key_1               : BOOL;                 (* 数字键1 *)
    Key_2               : BOOL;                 (* 数字键2 *)
    Key_3               : BOOL;                 (* 数字键3 *)
    Key_4               : BOOL;                 (* 数字键4 *)
    Key_5               : BOOL;                 (* 数字键5 *)
    Key_6               : BOOL;                 (* 数字键6 *)
    Key_7               : BOOL;                 (* 数字键7 *)
    Key_8               : BOOL;                 (* 数字键8 *)
    Key_9               : BOOL;                 (* 数字键9 *)
    Key_Clear           : BOOL;                 (* 清除键 (*) *)
    Key_Enter           : BOOL;                 (* 确认键 (#) *)
    Reset_Lock          : BOOL;                 (* 管理员解锁复位 *)
    Password_Single     : INT := 1504;          (* 单门密码 *)
    Password_Dual       : INT := 2502;          (* 双门密码 *)
    Max_Attempts        : INT := 3;             (* 最大尝试次数 *)
END_VAR

VAR_OUTPUT
    Single_Gate_Access  : BOOL;                 (* 单门访问权限 *)
    Dual_Gate_Access    : BOOL;                 (* 双门访问权限 *)
    Input_Active        : BOOL;                 (* 正在输入状态 *)
    System_Locked       : BOOL;                 (* 系统锁定状态 *)
    Error_Display       : BOOL;                 (* 错误显示 *)
    Input_Display       : STRING[4];           (* 输入显示（****） *)
    Status_Display      : STRING[20];          (* 状态显示信息 *)
    Attempts_Remaining  : INT;                  (* 剩余尝试次数 *)
END_VAR

VAR
    (* 密码输入缓冲区 *)
    Input_Buffer        : ARRAY[1..4] OF INT;  (* 输入缓冲区 *)
    Input_Index         : INT := 0;            (* 输入位置索引 *)
    Input_Password      : INT;                 (* 输入的完整密码 *)

    (* 按键边沿检测 *)
    Key_0_Last          : BOOL;
    Key_1_Last          : BOOL;
    Key_2_Last          : BOOL;
    Key_3_Last          : BOOL;
    Key_4_Last          : BOOL;
    Key_5_Last          : BOOL;
    Key_6_Last          : BOOL;
    Key_7_Last          : BOOL;
    Key_8_Last          : BOOL;
    Key_9_Last          : BOOL;
    Key_Clear_Last      : BOOL;
    Key_Enter_Last      : BOOL;
    Key_Edge_0          : BOOL;
    Key_Edge_1          : BOOL;
    Key_Edge_2          : BOOL;
    Key_Edge_3          : BOOL;
    Key_Edge_4          : BOOL;
    Key_Edge_5          : BOOL;
    Key_Edge_6          : BOOL;
    Key_Edge_7          : BOOL;
    Key_Edge_8          : BOOL;
    Key_Edge_9          : BOOL;
    Key_Edge_Clear      : BOOL;
    Key_Edge_Enter      : BOOL;

    (* 状态管理 *)
    Failed_Attempts     : INT := 0;            (* 失败尝试次数 *)
    Password_Valid      : BOOL;                (* 密码验证有效 *)
    Access_Type         : INT;                 (* 访问类型：1=单门，2=双门 *)

    (* 内部标志 *)
    Key_Pressed         : BOOL;                (* 按键按下标志 *)
    Pressed_Key         : INT;                 (* 按下的键值 *)
    Reset_Edge          : BOOL;                (* 复位边沿检测 *)
    Reset_Lock_Last     : BOOL;                (* 复位锁定前一周期状态 *)

    (* 显示相关 *)
    i                   : INT;                 (* 循环计数器 *)
    Error_Pulse         : BOOL;                (* 错误显示脉冲 *)
END_VAR

(* ============================================================================
   边沿检测器 - 基础变量实现R_TRIG
   ============================================================================ *)

Reset_Edge := Reset_Lock AND NOT Reset_Lock_Last;
Reset_Lock_Last := Reset_Lock;

(* 按键边沿检测 *)
Key_Edge_0 := Key_0 AND NOT Key_0_Last;
Key_0_Last := Key_0;

Key_Edge_1 := Key_1 AND NOT Key_1_Last;
Key_1_Last := Key_1;

Key_Edge_2 := Key_2 AND NOT Key_2_Last;
Key_2_Last := Key_2;

Key_Edge_3 := Key_3 AND NOT Key_3_Last;
Key_3_Last := Key_3;

Key_Edge_4 := Key_4 AND NOT Key_4_Last;
Key_4_Last := Key_4;

Key_Edge_5 := Key_5 AND NOT Key_5_Last;
Key_5_Last := Key_5;

Key_Edge_6 := Key_6 AND NOT Key_6_Last;
Key_6_Last := Key_6;

Key_Edge_7 := Key_7 AND NOT Key_7_Last;
Key_7_Last := Key_7;

Key_Edge_8 := Key_8 AND NOT Key_8_Last;
Key_8_Last := Key_8;

Key_Edge_9 := Key_9 AND NOT Key_9_Last;
Key_9_Last := Key_9;

Key_Edge_Clear := Key_Clear AND NOT Key_Clear_Last;
Key_Clear_Last := Key_Clear;

Key_Edge_Enter := Key_Enter AND NOT Key_Enter_Last;
Key_Enter_Last := Key_Enter;

(* ============================================================================
   系统锁定管理 - 简化版
   ============================================================================ *)

(* 锁定状态更新 *)
IF Failed_Attempts >= Max_Attempts THEN
    System_Locked := TRUE;
END_IF;

(* 锁定解除条件 *)
IF Reset_Edge THEN
    System_Locked := FALSE;
    Failed_Attempts := 0;
END_IF;

(* 计算剩余尝试次数 *)
Attempts_Remaining := Max_Attempts - Failed_Attempts;

(* ============================================================================
   按键处理逻辑
   ============================================================================ *)

Key_Pressed := FALSE;
Pressed_Key := -1;

(* 检测按下的数字键 *)
IF Key_Edge_0 THEN Key_Pressed := TRUE; Pressed_Key := 0; END_IF;
IF Key_Edge_1 THEN Key_Pressed := TRUE; Pressed_Key := 1; END_IF;
IF Key_Edge_2 THEN Key_Pressed := TRUE; Pressed_Key := 2; END_IF;
IF Key_Edge_3 THEN Key_Pressed := TRUE; Pressed_Key := 3; END_IF;
IF Key_Edge_4 THEN Key_Pressed := TRUE; Pressed_Key := 4; END_IF;
IF Key_Edge_5 THEN Key_Pressed := TRUE; Pressed_Key := 5; END_IF;
IF Key_Edge_6 THEN Key_Pressed := TRUE; Pressed_Key := 6; END_IF;
IF Key_Edge_7 THEN Key_Pressed := TRUE; Pressed_Key := 7; END_IF;
IF Key_Edge_8 THEN Key_Pressed := TRUE; Pressed_Key := 8; END_IF;
IF Key_Edge_9 THEN Key_Pressed := TRUE; Pressed_Key := 9; END_IF;

(* ============================================================================
   密码输入处理
   ============================================================================ *)

(* 只有在系统使能且未锁定时才能输入 *)
IF Enable AND NOT System_Locked THEN

    (* 清除键处理 *)
    IF Key_Edge_Clear THEN
        Input_Index := 0;
        FOR i := 1 TO 4 DO
            Input_Buffer[i] := 0;
        END_FOR;
        Input_Active := FALSE;
        Password_Valid := FALSE;
        Single_Gate_Access := FALSE;
        Dual_Gate_Access := FALSE;
        Error_Display := FALSE;
    END_IF;

    (* 数字键输入处理 *)
    IF Key_Pressed AND Pressed_Key >= 0 AND Pressed_Key <= 9 THEN
        Input_Active := TRUE;
        Error_Display := FALSE;

        IF Input_Index < 4 THEN
            Input_Index := Input_Index + 1;
            Input_Buffer[Input_Index] := Pressed_Key;
        END_IF;
    END_IF;

    (* 确认键处理 *)
    IF Key_Edge_Enter AND Input_Index = 4 THEN
        (* 计算输入的密码 *)
        Input_Password := Input_Buffer[1] * 1000 +
                         Input_Buffer[2] * 100 +
                         Input_Buffer[3] * 10 +
                         Input_Buffer[4];

        (* 密码验证 *)
        IF Input_Password = Password_Single THEN
            (* 单门密码正确 *)
            Access_Type := 1;
            Password_Valid := TRUE;
            Single_Gate_Access := TRUE;
            Dual_Gate_Access := FALSE;
            Failed_Attempts := 0;
            Error_Display := FALSE;
        ELSIF Input_Password = Password_Dual THEN
            (* 双门密码正确 *)
            Access_Type := 2;
            Password_Valid := TRUE;
            Single_Gate_Access := FALSE;
            Dual_Gate_Access := TRUE;
            Failed_Attempts := 0;
            Error_Display := FALSE;
        ELSE
            (* 密码错误 *)
            Password_Valid := FALSE;
            Single_Gate_Access := FALSE;
            Dual_Gate_Access := FALSE;
            Failed_Attempts := Failed_Attempts + 1;
            Error_Display := TRUE;
        END_IF;

        (* 清除输入缓冲区 *)
        Input_Index := 0;
        FOR i := 1 TO 4 DO
            Input_Buffer[i] := 0;
        END_FOR;
        Input_Active := FALSE;
    END_IF;

END_IF;

(* ============================================================================
   访问权限管理 - 简化版（权限立即生效，用户手动清除）
   ============================================================================ *)

(* 权限在密码正确后保持有效，直到用户清除或系统禁用 *)
IF NOT Enable OR Key_Edge_Clear THEN
    Single_Gate_Access := FALSE;
    Dual_Gate_Access := FALSE;
    Password_Valid := FALSE;
    Access_Type := 0;
END_IF;

(* ============================================================================
   显示处理
   ============================================================================ *)

(* 生成输入显示（星号掩码） *)
Input_Display := '';
FOR i := 1 TO Input_Index DO
    Input_Display := CONCAT(Input_Display, '*');
END_FOR;

(* 状态显示信息 *)
IF NOT Enable THEN
    Status_Display := 'SYSTEM DISABLED';
ELSIF System_Locked THEN
    Status_Display := 'SYSTEM LOCKED';
ELSIF Error_Display THEN
    Status_Display := 'INVALID PASSWORD';
ELSIF Input_Active THEN
    Status_Display := 'ENTER PASSWORD';
ELSIF Single_Gate_Access THEN
    Status_Display := 'SINGLE GATE ACCESS';
ELSIF Dual_Gate_Access THEN
    Status_Display := 'DUAL GATE ACCESS';
ELSE
    Status_Display := 'READY';
END_IF;

(* ============================================================================
   系统未使能时的处理
   ============================================================================ *)

IF NOT Enable THEN
    (* 清除所有状态 *)
    Input_Index := 0;
    Input_Active := FALSE;
    Password_Valid := FALSE;
    Single_Gate_Access := FALSE;
    Dual_Gate_Access := FALSE;
    Error_Display := FALSE;

    (* 清除输入缓冲区 *)
    FOR i := 1 TO 4 DO
        Input_Buffer[i] := 0;
    END_FOR;
END_IF;

END_FUNCTION_BLOCK

(* ---- DFB_Safety_Check.st ---- *)
(*
===============================================================================
DFB: DB_Safety_Check - 安全检测模块 (简化版)
===============================================================================
功能描述：
- 障碍物检测（光栅传感器）
- 过流保护检测
- 电源故障检测
- 安全状态综合判断
- 提供安全联锁信号

简化说明：
- 删除所有定时器和TIME类型变量
- 删除System_Clock输入
- 保留边沿检测（用基础BOOL实现）
- 保留核心的状态机和逻辑判断
- 即时响应安全检测，无延时过滤

作者: Claude Code Assistant
日期: 2025-09-24
版本: 2.0 (简化版)
===============================================================================
*)

FUNCTION_BLOCK DB_Safety_Check

VAR_INPUT
    Enable              : BOOL;         (* 系统使能 *)
    Passage_Sensor      : BOOL;         (* 通道光栅传感器（Bar_Lumineuse） *)
    Overcurrent_V1      : BOOL;         (* 门板1过流检测 *)
    Overcurrent_V2      : BOOL;         (* 门板2过流检测 *)
    Power_Loss_Alarm    : BOOL;         (* 市电故障报警 *)
    Gate1_Moving        : BOOL;         (* 门板1正在运动 *)
    Gate2_Moving        : BOOL;         (* 门板2正在运动 *)
    Safety_Reset        : BOOL;         (* 安全复位按钮 *)
END_VAR

VAR_OUTPUT
    Safe_To_Operate     : BOOL;         (* 安全运行许可 *)
    Obstacle_Detected   : BOOL;         (* 障碍物检测 *)
    Overcurrent_Gate1   : BOOL;         (* 门板1过流故障 *)
    Overcurrent_Gate2   : BOOL;         (* 门板2过流故障 *)
    Power_Fault         : BOOL;         (* 电源故障 *)
    Emergency_Stop      : BOOL;         (* 紧急停止输出 *)
    Reverse_Gate1       : BOOL;         (* 门板1反向命令 *)
    Reverse_Gate2       : BOOL;         (* 门板2反向命令 *)
    Safety_Warning      : BOOL;         (* 安全警告 *)
    Error_Code          : INT;          (* 安全错误代码 *)
END_VAR

VAR
    (* 安全复位边沿检测 *)
    Safety_Reset_Last   : BOOL;         (* 安全复位前一周期状态 *)
    Safety_Reset_Edge   : BOOL;         (* 安全复位边沿检测结果 *)

    (* 内部安全状态 *)
    Gate_Area_Occupied  : BOOL;         (* 门区域被占用 *)
    Overall_Safety      : BOOL;         (* 总体安全状态 *)

    (* 故障状态锁存 *)
    Overcurrent_Latched_V1 : BOOL;      (* 门板1过流锁存 *)
    Overcurrent_Latched_V2 : BOOL;      (* 门板2过流锁存 *)
    Power_Fault_Latched    : BOOL;      (* 电源故障锁存 *)
END_VAR

(* ============================================================================
   边沿检测器 - 基础变量实现R_TRIG
   ============================================================================ *)

Safety_Reset_Edge := Safety_Reset AND NOT Safety_Reset_Last;
Safety_Reset_Last := Safety_Reset;

(* ============================================================================
   障碍物检测逻辑 - 即时检测
   ============================================================================ *)

(* 通道传感器反向逻辑（光栅被遮挡时为FALSE） *)
Gate_Area_Occupied := NOT Passage_Sensor;

(* 即时障碍物检测（仅在门板运动时检测） *)
Obstacle_Detected := Gate_Area_Occupied AND (Gate1_Moving OR Gate2_Moving);

(* ============================================================================
   过流检测逻辑 - 即时检测，带锁存功能
   ============================================================================ *)

(* 门板1过流检测 - 即时响应并锁存 *)
IF Overcurrent_V1 AND Gate1_Moving THEN
    Overcurrent_Latched_V1 := TRUE;
END_IF;

(* 门板2过流检测 - 即时响应并锁存 *)
IF Overcurrent_V2 AND Gate2_Moving THEN
    Overcurrent_Latched_V2 := TRUE;
END_IF;

(* 输出过流状态 *)
Overcurrent_Gate1 := Overcurrent_Latched_V1;
Overcurrent_Gate2 := Overcurrent_Latched_V2;

(* ============================================================================
   反向控制逻辑（防夹保护） - 即时反向
   ============================================================================ *)

(* 检测到过流时立即反向 *)
Reverse_Gate1 := Overcurrent_Gate1;
Reverse_Gate2 := Overcurrent_Gate2;

(* ============================================================================
   电源故障检测 - 即时检测，带锁存功能
   ============================================================================ *)

(* 电源故障即时检测并锁存 *)
IF Power_Loss_Alarm THEN
    Power_Fault_Latched := TRUE;
END_IF;

Power_Fault := Power_Fault_Latched;

(* ============================================================================
   综合安全状态判断
   ============================================================================ *)

(* 计算总体安全状态 *)
Overall_Safety := Enable AND
                  NOT Obstacle_Detected AND
                  NOT Power_Fault AND
                  NOT Overcurrent_Gate1 AND
                  NOT Overcurrent_Gate2;

(* 安全运行许可 *)
Safe_To_Operate := Overall_Safety;

(* 紧急停止输出（任何安全条件不满足时激活） *)
Emergency_Stop := NOT Overall_Safety;

(* 安全警告（检测到潜在危险） *)
Safety_Warning := Gate_Area_Occupied OR
                  (Overcurrent_V1 AND NOT Overcurrent_Gate1) OR
                  (Overcurrent_V2 AND NOT Overcurrent_Gate2) OR
                  (Power_Loss_Alarm AND NOT Power_Fault);

(* ============================================================================
   错误代码生成
   ============================================================================ *)

(* 根据安全状态生成相应的错误代码 *)
IF NOT Enable THEN
    Error_Code := 2001;     (* 系统未使能 *)
ELSIF Obstacle_Detected THEN
    Error_Code := 2002;     (* 障碍物检测 *)
ELSIF Overcurrent_Gate1 THEN
    Error_Code := 2003;     (* 门板1过流 *)
ELSIF Overcurrent_Gate2 THEN
    Error_Code := 2004;     (* 门板2过流 *)
ELSIF Power_Fault THEN
    Error_Code := 2005;     (* 电源故障 *)
ELSE
    Error_Code := 0;        (* 无故障 *)
END_IF;

(* ============================================================================
   安全复位处理
   ============================================================================ *)

(* 当安全复位按钮按下且故障条件已清除时，允许复位 *)
IF Safety_Reset_Edge THEN
    (* 复位可恢复的故障状态 *)
    IF NOT Gate_Area_Occupied THEN
        (* 障碍物清除后自动复位，无需手动复位 *)
    END_IF;

    IF NOT Overcurrent_V1 THEN
        Overcurrent_Latched_V1 := FALSE;
    END_IF;

    IF NOT Overcurrent_V2 THEN
        Overcurrent_Latched_V2 := FALSE;
    END_IF;

    (* 电源故障需要故障源清除后才能复位 *)
    IF NOT Power_Loss_Alarm THEN
        Power_Fault_Latched := FALSE;
    END_IF;
END_IF;

(* ============================================================================
   系统未使能时的处理
   ============================================================================ *)

IF NOT Enable THEN
    (* 清除锁存的故障状态 *)
    Overcurrent_Latched_V1 := FALSE;
    Overcurrent_Latched_V2 := FALSE;
    Power_Fault_Latched := FALSE;
END_IF;

END_FUNCTION_BLOCK

(* ---- DFB_United_Control_Logic.st ---- *)
(*
===============================================================================
DFB: DB_United_Control_Logic - 统一门控制命令逻辑模块
===============================================================================
功能描述：
- 统一处理单门和双门的命令逻辑
- 处理遥控/键盘命令（cmd_v1_tele_digi, cmd_v12_tele_digi）
- 处理对讲命令（cmd_v1_interphone, cmd_v12_interphone）
- 根据Gate_Control DFB的状态输出相应的开关命令
- 控制辅助设备（警告灯、区域照明）

控制逻辑：
单门模式（V1）：
- 门关状态 + 单门命令 → 输出门1开启命令
- 门开状态 + 单门命令 → 输出门1关闭命令
- 门运动状态 + 单门命令 → 输出门1关闭命令

双门模式（V12）：
- 两门全关 + 双门命令 → 输出两门开启命令
- 两门全开 + 双门命令 → 输出两门关闭命令
- 混合/运动状态 + 双门命令 → 输出两门关闭命令

对讲模式：
- cmd_v1_interphone：作用等同于cmd_v1_tele_digi
- cmd_v12_interphone：作用等同于cmd_v12_tele_digi

输入参数：
- Enable: 系统使能信号
- cmd_v1_tele_digi: 单门遥控/键盘命令
- cmd_v12_tele_digi: 双门遥控/键盘命令
- cmd_v1_interphone: 单门对讲命令
- cmd_v12_interphone: 双门对讲命令
- Gate1_State: 门1状态（来自Gate_Control DFB）
- Gate2_State: 门2状态（来自Gate_Control DFB）

输出参数：
- Open_Command_V1: 门1开启命令输出
- Close_Command_V1: 门1关闭命令输出
- Open_Command_V2: 门2开启命令输出
- Close_Command_V2: 门2关闭命令输出
- Warning_Light: 警告灯输出
- Area_Light: 区域照明输出

作者: Claude Code Assistant
日期: 2025-09-24
版本: 2.0 (简化命令逻辑版)
===============================================================================
*)

FUNCTION_BLOCK DB_United_Control_Logic

VAR_INPUT
    Enable              : BOOL;     (* 系统使能信号 *)

    (* 命令输入信号 *)
    cmd_v1_tele_digi    : BOOL;     (* 单门遥控/键盘命令 *)
    cmd_v12_tele_digi   : BOOL;     (* 双门遥控/键盘命令 *)
    cmd_v1_interphone   : BOOL;     (* 单门对讲命令 *)
    cmd_v12_interphone  : BOOL;     (* 双门对讲命令 *)

    (* 门状态输入（来自Gate_Control DFB） *)
    Gate1_State         : INT;      (* 门1状态：0=关闭，1=开启中，2=开启，3=关闭中 *)
    Gate2_State         : INT;      (* 门2状态 *)
END_VAR

VAR_OUTPUT
    (* 门控制命令输出 *)
    Open_Command_V1     : BOOL;     (* 门1开启命令输出 *)
    Close_Command_V1    : BOOL;     (* 门1关闭命令输出 *)
    Open_Command_V2     : BOOL;     (* 门2开启命令输出 *)
    Close_Command_V2    : BOOL;     (* 门2关闭命令输出 *)

    (* 辅助设备输出 *)
    Warning_Light       : BOOL;     (* 警告灯输出 *)
    Area_Light          : BOOL;     (* 区域照明输出 *)
END_VAR

VAR
    (* 命令合并信号 *)
    cmd_v1_combined     : BOOL;     (* 单门命令合并（遥控+对讲） *)
    cmd_v12_combined    : BOOL;     (* 双门命令合并（遥控+对讲） *)

    (* 边沿检测变量 *)
    cmd_v1_prev         : BOOL := FALSE;
    cmd_v12_prev        : BOOL := FALSE;
    cmd_v1_edge         : BOOL;
    cmd_v12_edge        : BOOL;

    (* 状态判断变量 *)
    Gate1_Is_Open       : BOOL;
    Gate1_Is_Closed     : BOOL;
    Gate1_Is_Moving     : BOOL;
    Gate2_Is_Open       : BOOL;
    Gate2_Is_Closed     : BOOL;
    Gate2_Is_Moving     : BOOL;

    (* 双门组合状态 *)
    Both_Gates_Closed   : BOOL;
    Both_Gates_Open     : BOOL;
    Any_Gate_Moving     : BOOL;

    (* 双门延时控制 *)
    Dual_Open_Timer       : TIME := T#0S;    (* 双门开启延时计时器 *)
    Dual_Close_Timer      : TIME := T#0S;    (* 双门关闭延时计时器 *)
    Gate_Delay_Time       : TIME := T#1S;    (* 门间延时1秒 *)
    Scan_Time             : TIME := T#100MS; (* PLC扫描周期（假设100ms） *)

    (* 双门命令状态 *)
    Dual_Open_Active      : BOOL;     (* 双门开启过程激活 *)
    Dual_Close_Active     : BOOL;     (* 双门关闭过程激活 *)

    (* 延时完成标志 *)
    Dual_Open_Delay_Done  : BOOL;     (* 双门开启延时完成 *)
    Dual_Close_Delay_Done : BOOL;     (* 双门关闭延时完成 *)
END_VAR

(* ============================================================================ *)
(* 命令信号合并处理 *)
(* ============================================================================ *)

(* 单门命令合并：遥控/键盘 OR 对讲 *)
cmd_v1_combined := cmd_v1_tele_digi OR cmd_v1_interphone;

(* 双门命令合并：遥控/键盘 OR 对讲 *)
cmd_v12_combined := cmd_v12_tele_digi OR cmd_v12_interphone;

(* ============================================================================ *)
(* 边沿检测 *)
(* ============================================================================ *)

(* 单门命令边沿检测 *)
cmd_v1_edge := cmd_v1_combined AND NOT cmd_v1_prev;
cmd_v1_prev := cmd_v1_combined;

(* 双门命令边沿检测 *)
cmd_v12_edge := cmd_v12_combined AND NOT cmd_v12_prev;
cmd_v12_prev := cmd_v12_combined;

(* ============================================================================ *)
(* 门状态判断（基于输入的Gate_State） *)
(* ============================================================================ *)

(* 门1状态判断 *)
Gate1_Is_Closed := (Gate1_State = 0);    (* 0=关闭 *)
Gate1_Is_Open := (Gate1_State = 2);      (* 2=开启 *)
Gate1_Is_Moving := (Gate1_State = 1) OR (Gate1_State = 3);  (* 1=开启中，3=关闭中 *)

(* 门2状态判断 *)
Gate2_Is_Closed := (Gate2_State = 0);    (* 0=关闭 *)
Gate2_Is_Open := (Gate2_State = 2);      (* 2=开启 *)
Gate2_Is_Moving := (Gate2_State = 1) OR (Gate2_State = 3);  (* 1=开启中，3=关闭中 *)

(* 双门组合状态 *)
Both_Gates_Closed := Gate1_Is_Closed AND Gate2_Is_Closed;
Both_Gates_Open := Gate1_Is_Open AND Gate2_Is_Open;
Any_Gate_Moving := Gate1_Is_Moving OR Gate2_Is_Moving;

(* ============================================================================ *)
(* 双门延时控制逻辑 *)
(* ============================================================================ *)

(* 双门开启过程控制 *)
IF Dual_Open_Active THEN
    (* 立即启动门1 *)
    Open_Command_V1 := TRUE;

    (* 延时计时器递增 *)
    IF Dual_Open_Timer < Gate_Delay_Time THEN
        Dual_Open_Timer := Dual_Open_Timer + Scan_Time;
        Dual_Open_Delay_Done := FALSE;
    ELSE
        Dual_Open_Delay_Done := TRUE;
    END_IF;

    (* 延时完成后启动门2 *)
    IF Dual_Open_Delay_Done THEN
        Open_Command_V2 := TRUE;

        (* 当两门都开始运动或到达开启状态时，结束双门开启过程 *)
        IF (Gate1_Is_Moving OR Gate1_Is_Open) AND (Gate2_Is_Moving OR Gate2_Is_Open) THEN
            Dual_Open_Active := FALSE;
            Dual_Open_Timer := T#0S;
            Dual_Open_Delay_Done := FALSE;
        END_IF;
    END_IF;
END_IF;

(* 双门关闭过程控制 *)
IF Dual_Close_Active THEN
    (* 立即启动门2 *)
    Close_Command_V2 := TRUE;

    (* 延时计时器递增 *)
    IF Dual_Close_Timer < Gate_Delay_Time THEN
        Dual_Close_Timer := Dual_Close_Timer + Scan_Time;
        Dual_Close_Delay_Done := FALSE;
    ELSE
        Dual_Close_Delay_Done := TRUE;
    END_IF;

    (* 延时完成后启动门1 *)
    IF Dual_Close_Delay_Done THEN
        Close_Command_V1 := TRUE;

        (* 当两门都开始运动或到达关闭状态时，结束双门关闭过程 *)
        IF (Gate1_Is_Moving OR Gate1_Is_Closed) AND (Gate2_Is_Moving OR Gate2_Is_Closed) THEN
            Dual_Close_Active := FALSE;
            Dual_Close_Timer := T#0S;
            Dual_Close_Delay_Done := FALSE;
        END_IF;
    END_IF;
END_IF;

(* ============================================================================ *)
(* 命令逻辑处理 *)
(* ============================================================================ *)

(* 清除所有输出命令（如果不在延时控制过程中） *)
IF NOT Dual_Open_Active AND NOT Dual_Close_Active THEN
    Open_Command_V1 := FALSE;
    Close_Command_V1 := FALSE;
    Open_Command_V2 := FALSE;
    Close_Command_V2 := FALSE;
END_IF;

(* 只有在系统使能且检测到命令边沿时才处理 *)
IF Enable THEN

    (* 单门命令处理 *)
    IF cmd_v1_edge AND NOT Dual_Open_Active AND NOT Dual_Close_Active THEN
        IF Gate1_Is_Closed THEN
            (* 门1关闭状态：发出开门命令 *)
            Open_Command_V1 := TRUE;
        ELSIF Gate1_Is_Open THEN
            (* 门1开启状态：发出关门命令 *)
            Close_Command_V1 := TRUE;
        ELSIF Gate1_Is_Moving THEN
            (* 门1运动状态：发出关门命令（停止并关闭） *)
            Close_Command_V1 := TRUE;
        ELSE
            (* 未知状态：默认关门命令 *)
            Close_Command_V1 := TRUE;
        END_IF;
    END_IF;

    (* 双门命令处理 *)
    IF cmd_v12_edge AND NOT Dual_Open_Active AND NOT Dual_Close_Active THEN
        IF Both_Gates_Closed THEN
            (* 两门全关状态：启动双门开启过程 *)
            Dual_Open_Active := TRUE;
            Dual_Open_Timer := T#0S;      (* 重置计时器 *)
            Dual_Open_Delay_Done := FALSE;
        ELSIF Both_Gates_Open THEN
            (* 两门全开状态：启动双门关闭过程 *)
            Dual_Close_Active := TRUE;
            Dual_Close_Timer := T#0S;     (* 重置计时器 *)
            Dual_Close_Delay_Done := FALSE;
        ELSE
            (* 混合状态或运动状态：立即两门关闭 *)
            Close_Command_V1 := TRUE;
            Close_Command_V2 := TRUE;
        END_IF;
    END_IF;

END_IF;

(* ============================================================================ *)
(* 辅助设备控制 *)
(* ============================================================================ *)

(* 警告灯控制：任一门运动时点亮 *)
Warning_Light := Any_Gate_Moving;

(* 区域照明控制：有命令时点亮（简化版，只输出1） *)
Area_Light := cmd_v1_edge OR cmd_v12_edge;

(* ============================================================================ *)
(* 系统未使能时的安全处理 *)
(* ============================================================================ *)

IF NOT Enable THEN
    Open_Command_V1 := FALSE;
    Close_Command_V1 := FALSE;
    Open_Command_V2 := FALSE;
    Close_Command_V2 := FALSE;
    Warning_Light := FALSE;
END_IF;

END_FUNCTION_BLOCK

(* ---- DFB_Warning_Flash.st ---- *)
(*
===============================================================================
DFB: DFB_Warning_Flash - 警告灯闪烁控制模块
===============================================================================
功能描述：
- 当接收到持续的闪烁命令时，产生周期性的闪烁输出
- 支持可配置的闪烁频率和占空比
- 安全异常时（过流、通道有人）用于警告灯闪烁

输入参数：
- Enable: 系统使能信号
- Flash_Command: 闪烁命令（来自United_Control_Logic的Warning_Light）
- Flash_Period: 闪烁周期（PLC扫描周期数，默认500=约500ms）
- Duty_Cycle: 占空比（百分比，默认50%）

输出参数：
- Warning_Light_Out: 警告灯物理输出（连接到%Q0.3.4）

工作原理：
- Flash_Command=FALSE: 警告灯关闭
- Flash_Command=TRUE: 警告灯按设定频率闪烁

作者: Claude Code Assistant
日期: 2025-09-25
版本: 1.0
===============================================================================
*)

FUNCTION_BLOCK DFB_Warning_Flash

VAR_INPUT
    Enable          : BOOL := TRUE;     (* 系统使能信号 *)
    Flash_Command   : BOOL;             (* 闪烁命令信号 *)
    Flash_Period    : INT := 500;       (* 闪烁周期（PLC周期数） *)
    Duty_Cycle      : INT := 50;        (* 占空比（百分比） *)
END_VAR

VAR_OUTPUT
    Warning_Light_Out : BOOL;           (* 警告灯物理输出 *)
END_VAR

VAR
    Flash_Counter   : INT := 0;         (* 闪烁计数器 *)
    On_Time         : INT;              (* 点亮时间 *)
    Flash_State     : BOOL := FALSE;    (* 当前闪烁状态 *)
END_VAR

(* ============================================================================ *)
(* 闪烁逻辑实现 *)
(* ============================================================================ *)

(* 计算点亮时间（基于占空比） *)
On_Time := (Flash_Period * Duty_Cycle) / 100;

(* 系统使能且有闪烁命令时才工作 *)
IF Enable AND Flash_Command THEN

    (* 闪烁计数器递增 *)
    Flash_Counter := Flash_Counter + 1;

    (* 根据计数器位置决定闪烁状态 *)
    IF Flash_Counter <= On_Time THEN
        Flash_State := TRUE;        (* 点亮阶段 *)
    ELSE
        Flash_State := FALSE;       (* 熄灭阶段 *)
    END_IF;

    (* 周期结束，重置计数器 *)
    IF Flash_Counter >= Flash_Period THEN
        Flash_Counter := 0;
    END_IF;

    (* 输出闪烁状态 *)
    Warning_Light_Out := Flash_State;

ELSE
    (* 没有闪烁命令或系统未使能，关闭警告灯 *)
    Warning_Light_Out := FALSE;
    Flash_Counter := 0;
    Flash_State := FALSE;
END_IF;

END_FUNCTION_BLOCK

(* ---- MAIN_Program.st ---- *)
(*
===============================================================================
主控制程序 - MAIN
===============================================================================
功能描述：
这是双摆门控制系统的主控制程序，集成了所有功能模块：
- 双门板控制（单门/双门模式）
- 多种控制方式（遥控器、键盘、对讲机）
- 安全保护系统
- 照明和信号灯控制
- 故障诊断和报警

系统架构：
1. 安全检测模块 (Safety_Check)
2. 密码验证模块 (Keypad_Validation)
3. 命令管理模块 (Command_Manager)
4. 门板控制模块 (Gate1_Control, Gate2_Control)
5. 辅助设备控制（照明、信号灯）

I/O地址映射（基于CLAUDE.md）：
输出：
- %Q0.3.0: 门板1开启命令
- %Q0.3.1: 门板1关闭命令
- %Q0.3.2: 门板2开启命令
- %Q0.3.3: 门板2关闭命令
- %Q0.3.4: 警告信号灯
- %Q0.3.5: 区域照明

输入：
- %I0.2.0: 通道光栅传感器
- %I0.2.1: 门板2全开传感器
- %I0.2.2: 门板1全开传感器
- %I0.2.3: 门板1全关传感器
- %I0.2.4: 门板2全关传感器
- %I0.2.5: 门板2过流传感器
- %I0.2.6: 门板1过流传感器
- %I0.2.7: 对讲机单门命令
- %I0.2.8: 对讲机双门命令
- %I0.2.9: 遥控/键盘单门命令
- %I0.2.10: 遥控/键盘双门命令
- %I0.2.11: 市电故障报警

作者: Claude Code Assistant
日期: 2025-09-23
版本: 1.0
===============================================================================
*)

PROGRAM MAIN

VAR
    (*  ======================================================================== *)
    (*  系统控制变量 *)
    (*  ======================================================================== *)
    System_Enable           : BOOL := TRUE;     (*  系统总使能 *)
    First_Scan              : BOOL := TRUE;     (*  首次扫描标志 *)
    System_Ready            : BOOL;             (*  系统就绪状态 *)
    Emergency_Stop_Global   : BOOL;             (*  全局紧急停止 *)

    (*  ======================================================================== *)
    (* I/O映射变量（根据CLAUDE.md配置） *)
    (*  ======================================================================== *)

    (*  输入信号映射 *)
    Passage_Sensor          AT %I0.2.0  : BOOL; (*  通道光栅传感器 *)
    Gate2_Sensor_Open       AT %I0.2.1  : BOOL; (*  门板2全开传感器 *)
    Gate1_Sensor_Open       AT %I0.2.2  : BOOL; (*  门板1全开传感器 *)
    Gate1_Sensor_Close      AT %I0.2.3  : BOOL; (*  门板1全关传感器 *)
    Gate2_Sensor_Close      AT %I0.2.4  : BOOL; (*  门板2全关传感器 *)
    Gate2_Overcurrent       AT %I0.2.5  : BOOL; (*  门板2过流传感器 *)
    Gate1_Overcurrent       AT %I0.2.6  : BOOL; (*  门板1过流传感器 *)
    Intercom_Single_Cmd     AT %I0.2.7  : BOOL; (*  对讲机单门命令 *)
    Intercom_Dual_Cmd       AT %I0.2.8  : BOOL; (*  对讲机双门命令 *)
    Remote_Single_Cmd       AT %I0.2.9  : BOOL; (* 遥控/键盘单门命令 *)
    Remote_Dual_Cmd         AT %I0.2.10 : BOOL; (* 遥控/键盘双门命令 *)
    Power_Loss_Alarm        AT %I0.2.11 : BOOL; (*  市电故障报警 *)

    (*  输出信号映射 *)
    Gate1_Motor_Open        AT %Q0.3.0  : BOOL; (*  门板1开启命令 *)
    Gate1_Motor_Close       AT %Q0.3.1  : BOOL; (*  门板1关闭命令 *)
    Gate2_Motor_Open        AT %Q0.3.2  : BOOL; (*  门板2开启命令 *)
    Gate2_Motor_Close       AT %Q0.3.3  : BOOL; (*  门板2关闭命令 *)
    Warning_Light           AT %Q0.3.4  : BOOL; (*  警告信号灯 *)
    Area_Lighting           AT %Q0.3.5  : BOOL; (*  区域照明 *)

    (*  ======================================================================== *)
    (*  功能模块实例 *)
    (*  ======================================================================== *)

    (*  安全检测模块 *)
    Safety_Check            : DB_Safety_Check;

    (*  密码验证模块 *)
    Keypad_Validation       : DB_Keypad_Validation;

    (*  命令管理模块 *)
    Command_Manager         : DB_Command_Manager;

    (*  门板控制模块 *)
    Gate1_Control           : DB_Gate_Control;
    Gate2_Control           : DB_Gate_Control;

    (*  ======================================================================== *)
    (*  键盘接口变量（模拟键盘输入，实际应用中需要硬件接口） *)
    (*  ======================================================================== *)
    Keypad_Key_0            : BOOL; (*  数字键0-9 *)
    Keypad_Key_1            : BOOL;
    Keypad_Key_2            : BOOL;
    Keypad_Key_3            : BOOL;
    Keypad_Key_4            : BOOL;
    Keypad_Key_5            : BOOL;
    Keypad_Key_6            : BOOL;
    Keypad_Key_7            : BOOL;
    Keypad_Key_8            : BOOL;
    Keypad_Key_9            : BOOL;
    Keypad_Key_Clear        : BOOL; (*  清除键* *)
    Keypad_Key_Enter        : BOOL; (*  确认键# *)

    (*  ======================================================================== *)
    (*  系统状态和诊断变量 *)
    (*  ======================================================================== *)
    System_Status           : INT;   (*  系统状态：0=停止，1=运行，2=故障 *)
    Total_Error_Count       : INT;   (*  总错误计数 *)
    Last_Operation_Time     : TIME;  (*  最后操作时间 *)
    Operation_Counter       : DINT;  (*  操作计数器 *)

    (*  ======================================================================== *)
    (*  照明和信号控制变量 *)
    (*  ======================================================================== *)
    Lighting_Timer          : TON;   (*  照明延时关闭定时器 *)
    Lighting_Delay          : TIME := T#5m;    (*  照明延时时间 *)
    Warning_Blink_Timer     : TOF;   (*  警告灯闪烁定时器 *)
    Warning_Blink_Cycle     : TIME := T#500ms; (*  闪烁周期 *)

    (*  ======================================================================== *)
    (*  内部连接变量 *)
    (*  ======================================================================== *)
    Safety_Status           : BOOL;  (*  安全状态 *)
    Command_Valid           : BOOL;  (*  命令有效 *)
    Gate1_Moving            : BOOL;  (*  门板1运动状态 *)
    Gate2_Moving            : BOOL;  (*  门板2运动状态 *)
    Any_Gate_Moving         : BOOL;  (*  任意门板运动 *)
    Keypad_Access_Single    : BOOL;  (*  键盘单门权限 *)
    Keypad_Access_Dual      : BOOL;  (*  键盘双门权限 *)
END_VAR

(*  ============================================================================ *)
(*  系统初始化 *)
(*  ============================================================================ *)

IF First_Scan THEN
    (*  系统启动初始化 *)
    System_Enable := TRUE;
    System_Status := 0; (*  系统停止状态 *)
    Total_Error_Count := 0;
    Operation_Counter := 0;

    (*  输出安全状态 *)
    Gate1_Motor_Open := FALSE;
    Gate1_Motor_Close := FALSE;
    Gate2_Motor_Open := FALSE;
    Gate2_Motor_Close := FALSE;
    Warning_Light := FALSE;
    Area_Lighting := FALSE;

    First_Scan := FALSE;
END_IF;

(*  ============================================================================ *)
(*  安全检测模块 *)
(*  ============================================================================ *)

Safety_Check(
    Enable := System_Enable,
    Passage_Sensor := Passage_Sensor,
    Overcurrent_V1 := Gate1_Overcurrent,
    Overcurrent_V2 := Gate2_Overcurrent,
    Power_Loss_Alarm := Power_Loss_Alarm,
    Gate1_Moving := Gate1_Moving,
    Gate2_Moving := Gate2_Moving,
    Safety_Reset := FALSE (*  可以连接到维护面板的复位按钮 *)
);

(*  获取安全状态 *)
Safety_Status := Safety_Check.Safe_To_Operate;
Emergency_Stop_Global := Safety_Check.Emergency_Stop;

(*  ============================================================================ *)
(*  密码验证模块（键盘接口） *)
(*  ============================================================================ *)

(*  注意：实际应用中需要通过FBD连接键盘扫描电路 *)
(*  这里提供了接口变量，需要在FBD中实现键盘扫描逻辑 *)

Keypad_Validation(
    Enable := System_Enable,
    Key_0 := Keypad_Key_0,
    Key_1 := Keypad_Key_1,
    Key_2 := Keypad_Key_2,
    Key_3 := Keypad_Key_3,
    Key_4 := Keypad_Key_4,
    Key_5 := Keypad_Key_5,
    Key_6 := Keypad_Key_6,
    Key_7 := Keypad_Key_7,
    Key_8 := Keypad_Key_8,
    Key_9 := Keypad_Key_9,
    Key_Clear := Keypad_Key_Clear,
    Key_Enter := Keypad_Key_Enter,
    Reset_Lock := FALSE (*  可以连接到管理员复位按钮 *)
);

(*  获取键盘访问权限 *)
Keypad_Access_Single := Keypad_Validation.Single_Gate_Access;
Keypad_Access_Dual := Keypad_Validation.Dual_Gate_Access;

(*  ============================================================================ *)
(*  命令管理模块 *)
(*  ============================================================================ *)

Command_Manager(
    Enable := System_Enable,
    (* 遥控器/键盘命令（通过权限验证） *)
    Remote_Single_Gate := Remote_Single_Cmd,
    Remote_Dual_Gate := Remote_Dual_Cmd,
    Keypad_Single_Gate := Keypad_Access_Single,
    Keypad_Dual_Gate := Keypad_Access_Dual,
    (*  对讲机命令（直接连接） *)
    Intercom_Single_Gate := Intercom_Single_Cmd,
    Intercom_Dual_Gate := Intercom_Dual_Cmd,
    (*  安全状态 *)
    Safety_OK := Safety_Status,
    Gate1_Status_Closed := Gate1_Control.Status_Closed,
    Gate1_Status_Open := Gate1_Control.Status_Open,
    Gate2_Status_Closed := Gate2_Control.Status_Closed,
    Gate2_Status_Open := Gate2_Control.Status_Open
);

(*  获取命令状态 *)
Command_Valid := Command_Manager.Command_Valid;

(*  ============================================================================ *)
(*  门板1控制模块 *)
(*  ============================================================================ *)

Gate1_Control(
    Enable := System_Enable,
    Open_Cmd := Command_Manager.Gate1_Open_Command,
    Close_Cmd := Command_Manager.Gate1_Close_Command,
    Emergency_Stop := NOT Emergency_Stop_Global,
    Sensor_Open := Gate1_Sensor_Open,
    Sensor_Close := Gate1_Sensor_Close,
    Overcurrent := Gate1_Overcurrent OR Safety_Check.Overcurrent_Gate1,
    Max_Open_Time := T#25s,
    Max_Close_Time := T#25s
);

(*  获取门板1状态 *)
Gate1_Moving := Gate1_Control.Status_Opening OR Gate1_Control.Status_Closing;

(*  ============================================================================ *)
(*  门板2控制模块 *)
(*  ============================================================================ *)

Gate2_Control(
    Enable := System_Enable,
    Open_Cmd := Command_Manager.Gate2_Open_Command,
    Close_Cmd := Command_Manager.Gate2_Close_Command,
    Emergency_Stop := NOT Emergency_Stop_Global,
    Sensor_Open := Gate2_Sensor_Open,
    Sensor_Close := Gate2_Sensor_Close,
    Overcurrent := Gate2_Overcurrent OR Safety_Check.Overcurrent_Gate2,
    Max_Open_Time := T#25s,
    Max_Close_Time := T#25s
);

(*  获取门板2状态 *)
Gate2_Moving := Gate2_Control.Status_Opening OR Gate2_Control.Status_Closing;

(*  ============================================================================ *)
(*  电机输出控制 *)
(*  ============================================================================ *)

(*  门板1电机控制（带安全保护） *)
IF System_Enable AND NOT Emergency_Stop_Global THEN
    Gate1_Motor_Open := Gate1_Control.Motor_Open;
    Gate1_Motor_Close := Gate1_Control.Motor_Close;

    (*  防夹保护：过流时反向 *)
    IF Safety_Check.Reverse_Gate1 THEN
        IF Gate1_Control.Status_Opening THEN
            Gate1_Motor_Open := FALSE;
            Gate1_Motor_Close := TRUE;
        ELSIF Gate1_Control.Status_Closing THEN
            Gate1_Motor_Close := FALSE;
            Gate1_Motor_Open := TRUE;
        END_IF;
    END_IF;
ELSE
    Gate1_Motor_Open := FALSE;
    Gate1_Motor_Close := FALSE;
END_IF;

(*  门板2电机控制（带安全保护） *)
IF System_Enable AND NOT Emergency_Stop_Global THEN
    Gate2_Motor_Open := Gate2_Control.Motor_Open;
    Gate2_Motor_Close := Gate2_Control.Motor_Close;

    (*  防夹保护：过流时反向 *)
    IF Safety_Check.Reverse_Gate2 THEN
        IF Gate2_Control.Status_Opening THEN
            Gate2_Motor_Open := FALSE;
            Gate2_Motor_Close := TRUE;
        ELSIF Gate2_Control.Status_Closing THEN
            Gate2_Motor_Close := FALSE;
            Gate2_Motor_Open := TRUE;
        END_IF;
    END_IF;
ELSE
    Gate2_Motor_Open := FALSE;
    Gate2_Motor_Close := FALSE;
END_IF;

(*  ============================================================================ *)
(*  警告信号灯控制 *)
(*  ============================================================================ *)

Any_Gate_Moving := Gate1_Moving OR Gate2_Moving;

(*  警告灯闪烁控制 *)
Warning_Blink_Timer(
    IN := Any_Gate_Moving,
    PT := Warning_Blink_Cycle
);

(*  门板运动时警告灯闪烁，故障时常亮 *)
IF Any_Gate_Moving THEN
    Warning_Light := NOT Warning_Blink_Timer.Q; (*  闪烁 *)
ELSIF Safety_Check.Emergency_Stop OR
      Gate1_Control.Error OR
      Gate2_Control.Error THEN
    Warning_Light := TRUE; (*  故障时常亮 *)
ELSE
    Warning_Light := FALSE;
END_IF;

(*  ============================================================================ *)
(*  区域照明控制 *)
(*  ============================================================================ *)

(*  照明延时关闭定时器 *)
Lighting_Timer(
    IN := NOT (Any_Gate_Moving OR Command_Manager.Command_Active),
    PT := Lighting_Delay
);

(*  照明控制逻辑：有活动时开启，延时后关闭 *)
IF Any_Gate_Moving OR
   Command_Manager.Command_Active OR
   Safety_Check.Obstacle_Detected THEN
    Area_Lighting := TRUE;
ELSIF Lighting_Timer.Q THEN
    Area_Lighting := FALSE;
END_IF;

(*  ============================================================================ *)
(*  系统状态管理和诊断 *)
(*  ============================================================================ *)

(*  计算系统状态 *)
IF NOT System_Enable THEN
    System_Status := 0; (*  系统停止 *)
ELSIF Safety_Check.Emergency_Stop OR
      Gate1_Control.Error OR
      Gate2_Control.Error OR
      Keypad_Validation.System_Locked THEN
    System_Status := 2; (*  系统故障 *)
ELSE
    System_Status := 1; (*  系统正常运行 *)
END_IF;

(*  系统就绪状态 *)
System_Ready := (System_Status = 1) AND NOT Any_Gate_Moving;

(*  错误计数统计 *)
IF Gate1_Control.Error OR
   Gate2_Control.Error OR
   Safety_Check.Emergency_Stop THEN
    Total_Error_Count := Total_Error_Count + 1;
    (*  防止计数溢出 *)
    IF Total_Error_Count > 9999 THEN
        Total_Error_Count := 0;
    END_IF;
END_IF;

(*  操作计数（每次门操作） *)
IF Command_Manager.Command_Active THEN
    Operation_Counter := Operation_Counter + 1;
    Last_Operation_Time := TIME(); (*  需要系统时间函数支持 *)
    (*  防止计数溢出 *)
    IF Operation_Counter > 999999 THEN
        Operation_Counter := 0;
    END_IF;
END_IF;

(*  ============================================================================ *)
(*  系统关闭处理 *)
(*  ============================================================================ *)

IF NOT System_Enable THEN
    (*  安全关闭所有输出 *)
    Gate1_Motor_Open := FALSE;
    Gate1_Motor_Close := FALSE;
    Gate2_Motor_Open := FALSE;
    Gate2_Motor_Close := FALSE;
    Warning_Light := FALSE;
    Area_Lighting := FALSE;
END_IF;

END_PROGRAM

(*
===============================================================================
FBD 连接说明
===============================================================================

在Unity Pro中，需要在FBD（功能块图）中实现以下硬件接口连接：

1. 键盘扫描模块：
   - 使用矩阵键盘扫描FFB
   - 连接Keypad_Key_0到Keypad_Key_9变量
   - 连接Keypad_Key_Clear和Keypad_Key_Enter变量

2. 通信模块：
   - 如需远程监控，可添加以太网通信FFB
   - 连接到NOE 100.2模块（IP: 134.214.184.171）
   - 实现远程诊断和控制接口

3. HMI接口：
   - 连接人机界面显示模块
   - 显示系统状态、错误代码、操作计数等
   - 提供手动控制和参数设置界面

4. 数据记录：
   - 可选添加数据记录FFB
   - 记录操作历史、故障日志等

使用方法：
1. 在Unity Pro中创建新项目
2. 导入各个DFB文件
3. 创建MAIN程序并粘贴上述代码
4. 在FBD中添加必要的硬件接口连接
5. 配置I/O地址映射
6. 编译并下载到PLC

===============================================================================
*)
